LIN {X 0,Y 361.998,Z 160.89,A -85,B 0,C 180,E1 -12946.528,E2 -12946.528} C_VEL
LIN {X 0,Y 362.031,Z 160.886,A -85,B 0,C 180,E1 -12949.938,E2 -12949.938} C_VEL
LIN {X 0,Y 362.16,Z 160.873,A -85,B 0,C 180,E1 -12953.314,E2 -12953.314} C_VEL
LIN {X 0,Y 362.282,Z 160.854,A -85,B 0,C 180,E1 -12957.776,E2 -12957.776} C_VEL
LIN {X 0,Y 362.425,Z 160.836,A -85,B 0,C 180,E1 -12960,E2 -12960} C_VEL
LIN {X 0,Y 362.281,Z 160.856,A -85,B 0,C 180,E1 -12962.224,E2 -12962.224} C_VEL
LIN {X 0,Y 362.16,Z 160.875,A -85,B 0,C 180,E1 -12966.686,E2 -12966.686} C_VEL
LIN {X 0,Y 362.03,Z 160.888,A -85,B 0,C 180,E1 -12970.062,E2 -12970.062} C_VEL
LIN {X 0,Y 361.997,Z 160.891,A -85,B 0,C 180,E1 -12973.899,E2 -12973.899} C_VEL
LIN {X 0,Y 361.966,Z 160.896,A -85,B 0,C 180,E1 -12977.939,E2 -12977.939} C_VEL
LIN {X 0,Y 361.86,Z 160.908,A -85,B 0,C 180,E1 -12981.655,E2 -12981.655} C_VEL
LIN {X 0,Y 361.926,Z 160.899,A -85,B 0,C 180,E1 -12985.29,E2 -12985.29} C_VEL
LIN {X 0,Y 361.908,Z 160.905,A -85,B 0,C 180,E1 -12987.779,E2 -12987.779} C_VEL
LIN {X 0,Y 361.837,Z 160.913,A -85,B 0,C 180,E1 -12991.63,E2 -12991.63} C_VEL
LIN {X 0,Y 361.873,Z 160.907,A -85,B 0,C 180,E1 -12995.345,E2 -12995.345} C_VEL
LIN {X 0,Y 361.862,Z 160.907,A -85,B 0,C 180,E1 -12999.026,E2 -12999.026} C_VEL
LIN {X 0,Y 361.834,Z 160.911,A -85,B 0,C 180,E1 -13002.829,E2 -13002.829} C_VEL
LIN {X 0,Y 361.817,Z 160.914,A -85,B 0,C 180,E1 -13005.947,E2 -13005.947} C_VEL
LIN {X 0,Y 361.813,Z 160.918,A -85,B 0,C 180,E1 -13009.249,E2 -13009.249} C_VEL
LIN {X 0,Y 361.865,Z 160.91,A -85,B 0,C 180,E1 -13012.982,E2 -13012.982} C_VEL
LIN {X 0,Y 361.859,Z 160.909,A -85,B 0,C 180,E1 -13016.631,E2 -13016.631} C_VEL
LIN {X 0,Y 361.903,Z 160.997,A -85,B 0,C 180,E1 -13020.494,E2 -13020.494} C_VEL
LIN {X 0,Y 364.387,Z 172.887,A -85,B 0,C 180,E1 -13023.666,E2 -13023.666} C_VEL
LIN {X 0,Y 365.605,Z 180.414,A -85,B 0,C 180,E1 -13025.588,E2 -13025.588} C_VEL
LIN {X 0,Y 364.663,Z 190.236,A -85,B 0,C 180,E1 -13027.892,E2 -13027.892} C_VEL
LIN {X 0,Y 369.444,Z 217.539,A -85,B 0,C 180,E1 -13028.771,E2 -13028.771} C_VEL
LIN {X 0,Y 370.205,Z 224.641,A -85,B 0,C 180,E1 -13028.961,E2 -13028.961} C_VEL
LIN {X 0,Y 368.998,Z 298.645,A -85,B 0,C 180,E1 -13030.422,E2 -13030.422} C_VEL
LIN {X 0,Y 368.329,Z 311.846,A -85,B 0,C 180,E1 -13030.892,E2 -13030.892} C_VEL
LIN {X 0,Y 367.51,Z 323.969,A -85,B 0,C 180,E1 -13031.535,E2 -13031.535} C_VEL
LIN {X 0,Y 366.496,Z 336.205,A -85,B 0,C 180,E1 -13032.421,E2 -13032.421} C_VEL
LIN {X 0,Y 365.288,Z 347.782,A -85,B 0,C 180,E1 -13033.514,E2 -13033.514} C_VEL
LIN {X 0,Y 364.282,Z 357.893,A -85,B 0,C 180,E1 -13034.718,E2 -13034.718} C_VEL
LIN {X 0,Y 363.402,Z 366.737,A -85,B 0,C 180,E1 -13036.011,E2 -13036.011} C_VEL
LIN {X 0,Y 362.508,Z 374.603,A -85,B 0,C 180,E1 -13037.402,E2 -13037.402} C_VEL
LIN {X 0,Y 361.621,Z 382.284,A -85,B 0,C 180,E1 -13039.077,E2 -13039.077} C_VEL
LIN {X 0,Y 360.938,Z 389.371,A -85,B 0,C 180,E1 -13041.039,E2 -13041.039} C_VEL
LIN {X 0,Y 360.592,Z 394.086,A -85,B 0,C 180,E1 -13042.722,E2 -13042.722} C_VEL
LIN {X 0,Y 360.363,Z 397.689,A -85,B 0,C 180,E1 -13044.404,E2 -13044.404} C_VEL
LIN {X 0,Y 360.342,Z 399.548,A -85,B 0,C 180,E1 -13045.526,E2 -13045.526} C_VEL
LIN {X 0,Y 360.289,Z 400.941,A -85,B 0,C 180,E1 -13046.645,E2 -13046.645} C_VEL
LIN {X 0,Y 360.289,Z 402.543,A -85,B 0,C 180,E1 -13048.882,E2 -13048.882} C_VEL
LIN {X 0,Y 360.312,Z 402.757,A -85,B 0,C 180,E1 -13050,E2 -13050} C_VEL
LIN {X 0,Y 360.289,Z 402.538,A -85,B 0,C 180,E1 -13051.118,E2 -13051.118} C_VEL
LIN {X 0,Y 360.289,Z 400.931,A -85,B 0,C 180,E1 -13053.355,E2 -13053.355} C_VEL
LIN {X 0,Y 360.342,Z 399.533,A -85,B 0,C 180,E1 -13054.474,E2 -13054.474} C_VEL
LIN {X 0,Y 360.378,Z 396.969,A -85,B 0,C 180,E1 -13055.961,E2 -13055.961} C_VEL
LIN {X 0,Y 360.673,Z 392.619,A -85,B 0,C 180,E1 -13057.84,E2 -13057.84} C_VEL
LIN {X 0,Y 361.189,Z 386.507,A -85,B 0,C 180,E1 -13059.803,E2 -13059.803} C_VEL
LIN {X 0,Y 361.852,Z 379.831,A -85,B 0,C 180,E1 -13061.483,E2 -13061.483} C_VEL
LIN {X 0,Y 362.835,Z 371.552,A -85,B 0,C 180,E1 -13063.155,E2 -13063.155} C_VEL
LIN {X 0,Y 363.7,Z 363.06,A -85,B 0,C 180,E1 -13064.549,E2 -13064.549} C_VEL
LIN {X 0,Y 364.787,Z 352.569,A -85,B 0,C 180,E1 -13065.935,E2 -13065.935} C_VEL
LIN {X 0,Y 366.004,Z 340.762,A -85,B 0,C 180,E1 -13067.171,E2 -13067.171} C_VEL
LIN {X 0,Y 367.094,Z 328.878,A -85,B 0,C 180,E1 -13068.126,E2 -13068.126} C_VEL
LIN {X 0,Y 367.988,Z 316.508,A -85,B 0,C 180,E1 -13068.873,E2 -13068.873} C_VEL
LIN {X 0,Y 368.769,Z 303.791,A -85,B 0,C 180,E1 -13069.41,E2 -13069.41} C_VEL
LIN {X 0,Y 369.229,Z 290.405,A -85,B 0,C 180,E1 -13069.746,E2 -13069.746} C_VEL
LIN {X 0,Y 370.135,Z 222.324,A -85,B 0,C 180,E1 -13071.075,E2 -13071.075} C_VEL
LIN {X 0,Y 365.002,Z 192.189,A -85,B 0,C 180,E1 -13072.008,E2 -13072.008} C_VEL
LIN {X 0,Y 364.692,Z 190.305,A -85,B 0,C 180,E1 -13072.073,E2 -13072.073} C_VEL
LIN {X 0,Y 365.613,Z 180.345,A -85,B 0,C 180,E1 -13074.411,E2 -13074.411} C_VEL
LIN {X 0,Y 364.398,Z 172.814,A -85,B 0,C 180,E1 -13076.333,E2 -13076.333} C_VEL
LIN {X 0,Y 361.864,Z 160.906,A -85,B 0,C 180,E1 -13079.554,E2 -13079.554} C_VEL
LIN {X 0,Y 361.858,Z 160.909,A -85,B 0,C 180,E1 -13083.369,E2 -13083.369} C_VEL
LIN {X 0,Y 361.863,Z 160.911,A -85,B 0,C 180,E1 -13087.018,E2 -13087.018} C_VEL
LIN {X 0,Y 361.813,Z 160.919,A -85,B 0,C 180,E1 -13090.751,E2 -13090.751} C_VEL
LIN {X 0,Y 361.817,Z 160.916,A -85,B 0,C 180,E1 -13094.368,E2 -13094.368} C_VEL
LIN {X 0,Y 361.832,Z 160.91,A -85,B 0,C 180,E1 -13097.569,E2 -13097.569} C_VEL
LIN {X 0,Y 361.863,Z 160.908,A -85,B 0,C 180,E1 -13100.975,E2 -13100.975} C_VEL
LIN {X 0,Y 361.874,Z 160.908,A -85,B 0,C 180,E1 -13104.655,E2 -13104.655} C_VEL
LIN {X 0,Y 361.837,Z 160.914,A -85,B 0,C 180,E1 -13108.37,E2 -13108.37} C_VEL
LIN {X 0,Y 361.865,Z 160.906,A -85,B 0,C 180,E1 -13110.952,E2 -13110.952} C_VEL
LIN {X 0,Y 361.893,Z 160.903,A -85,B 0,C 180,E1 -13114.707,E2 -13114.707} C_VEL
LIN {X 0,Y 361.86,Z 160.909,A -85,B 0,C 180,E1 -13118.345,E2 -13118.345} C_VEL
LIN {X 0,Y 361.967,Z 160.896,A -85,B 0,C 180,E1 -13122.061,E2 -13122.061} C_VEL
LIN {X 0,Y 361.998,Z 160.891,A -85,B 0,C 180,E1 -13126.101,E2 -13126.101} C_VEL
LIN {X 0,Y 362.031,Z 160.888,A -85,B 0,C 180,E1 -13129.938,E2 -13129.938} C_VEL
LIN {X 0,Y 362.16,Z 160.874,A -85,B 0,C 180,E1 -13133.314,E2 -13133.314} C_VEL
LIN {X 0,Y 362.282,Z 160.856,A -85,B 0,C 180,E1 -13137.776,E2 -13137.776} C_VEL
LIN {X 0,Y 362.426,Z 160.836,A -85,B 0,C 180,E1 -13140,E2 -13140} C_VEL
LIN {X 0,Y 362.282,Z 160.854,A -85,B 0,C 180,E1 -13142.224,E2 -13142.224} C_VEL
LIN {X 0,Y 362.147,Z 160.874,A -85,B 0,C 180,E1 -13146.687,E2 -13146.687} C_VEL
LIN {X 0,Y 362.055,Z 160.889,A -85,B 0,C 180,E1 -13148.934,E2 -13148.934} C_VEL
LIN {X 0,Y 361.959,Z 160.896,A -85,B 0,C 180,E1 -13152.332,E2 -13152.332} C_VEL
LIN {X 0,Y 361.962,Z 160.898,A -85,B 0,C 180,E1 -13154.62,E2 -13154.62} C_VEL
LIN {X 0,Y 361.96,Z 160.895,A -85,B 0,C 180,E1 -13158.099,E2 -13158.099} C_VEL
LIN {X 0,Y 361.892,Z 160.903,A -85,B 0,C 180,E1 -13161.653,E2 -13161.653} C_VEL
LIN {X 0,Y 361.929,Z 160.898,A -85,B 0,C 180,E1 -13165.29,E2 -13165.29} C_VEL
LIN {X 0,Y 361.918,Z 160.9,A -85,B 0,C 180,E1 -13167.778,E2 -13167.778} C_VEL
LIN {X 0,Y 361.847,Z 160.908,A -85,B 0,C 180,E1 -13171.285,E2 -13171.285} C_VEL
LIN {X 0,Y 361.855,Z 160.913,A -85,B 0,C 180,E1 -13174.281,E2 -13174.281} C_VEL
LIN {X 0,Y 361.864,Z 160.906,A -85,B 0,C 180,E1 -13177.223,E2 -13177.223} C_VEL
LIN {X 0,Y 361.836,Z 160.91,A -85,B 0,C 180,E1 -13180.756,E2 -13180.756} C_VEL
LIN {X 0,Y 361.819,Z 160.914,A -85,B 0,C 180,E1 -13184.369,E2 -13184.369} C_VEL
LIN {X 0,Y 361.837,Z 160.913,A -85,B 0,C 180,E1 -13187.568,E2 -13187.568} C_VEL
LIN {X 0,Y 361.869,Z 160.906,A -85,B 0,C 180,E1 -13190.974,E2 -13190.974} C_VEL
LIN {X 0,Y 361.875,Z 160.905,A -85,B 0,C 180,E1 -13194.655,E2 -13194.655} C_VEL
LIN {X 0,Y 361.839,Z 160.91,A -85,B 0,C 180,E1 -13198.371,E2 -13198.371} C_VEL
LIN {X 0,Y 361.902,Z 160.904,A -85,B 0,C 180,E1 -13200.955,E2 -13200.955} C_VEL
LIN {X 0,Y 361.99,Z 161.002,A -85,B 0,C 180,E1 -13204.059,E2 -13204.059} C_VEL
LIN {X 0,Y 364.077,Z 171.501,A -85,B 0,C 180,E1 -13206.99,E2 -13206.99} C_VEL
LIN {X 0,Y 364.819,Z 175.438,A -85,B 0,C 180,E1 -13207.999,E2 -13207.999} C_VEL
LIN {X 0,Y 367.194,Z 184.857,A -85,B 0,C 180,E1 -13208.344,E2 -13208.344} C_VEL
LIN {X 0,Y 370.497,Z 201.339,A -85,B 0,C 180,E1 -13208.885,E2 -13208.885} C_VEL
LIN {X 0,Y 369.221,Z 281.969,A -85,B 0,C 180,E1 -13210.47,E2 -13210.47} C_VEL
LIN {X 0,Y 368.677,Z 295.427,A -85,B 0,C 180,E1 -13210.947,E2 -13210.947} C_VEL
LIN {X 0,Y 367.888,Z 308.218,A -85,B 0,C 180,E1 -13211.627,E2 -13211.627} C_VEL
LIN {X 0,Y 367.02,Z 319.572,A -85,B 0,C 180,E1 -13212.447,E2 -13212.447} C_VEL
LIN {X 0,Y 365.946,Z 331.168,A -85,B 0,C 180,E1 -13213.537,E2 -13213.537} C_VEL
LIN {X 0,Y 365.13,Z 340.627,A -85,B 0,C 180,E1 -13214.653,E2 -13214.653} C_VEL
LIN {X 0,Y 364.069,Z 350.244,A -85,B 0,C 180,E1 -13216.037,E2 -13216.037} C_VEL
LIN {X 0,Y 363.112,Z 358.121,A -85,B 0,C 180,E1 -13217.424,E2 -13217.424} C_VEL
LIN {X 0,Y 362.22,Z 365.819,A -85,B 0,C 180,E1 -13219.095,E2 -13219.095} C_VEL
LIN {X 0,Y 361.392,Z 372.884,A -85,B 0,C 180,E1 -13221.05,E2 -13221.05} C_VEL
LIN {X 0,Y 360.959,Z 377.589,A -85,B 0,C 180,E1 -13222.729,E2 -13222.729} C_VEL
LIN {X 0,Y 360.709,Z 381.189,A -85,B 0,C 180,E1 -13224.409,E2 -13224.409} C_VEL
LIN {X 0,Y 360.545,Z 383.05,A -85,B 0,C 180,E1 -13225.528,E2 -13225.528} C_VEL
LIN {X 0,Y 360.403,Z 384.452,A -85,B 0,C 180,E1 -13226.646,E2 -13226.646} C_VEL
LIN {X 0,Y 360.333,Z 386.061,A -85,B 0,C 180,E1 -13228.882,E2 -13228.882} C_VEL
LIN {X 0,Y 360.315,Z 386.294,A -85,B 0,C 180,E1 -13230,E2 -13230} C_VEL
LIN {X 0,Y 360.333,Z 386.104,A -85,B 0,C 180,E1 -13231.118,E2 -13231.118} C_VEL
LIN {X 0,Y 360.401,Z 384.552,A -85,B 0,C 180,E1 -13233.354,E2 -13233.354} C_VEL
LIN {X 0,Y 360.537,Z 383.194,A -85,B 0,C 180,E1 -13234.472,E2 -13234.472} C_VEL
LIN {X 0,Y 360.81,Z 379.409,A -85,B 0,C 180,E1 -13236.585,E2 -13236.585} C_VEL
LIN {X 0,Y 361.206,Z 374.877,A -85,B 0,C 180,E1 -13238.391,E2 -13238.391} C_VEL
LIN {X 0,Y 361.947,Z 368.434,A -85,B 0,C 180,E1 -13240.347,E2 -13240.347} C_VEL
LIN {X 0,Y 362.718,Z 361.356,A -85,B 0,C 180,E1 -13242.022,E2 -13242.022} C_VEL
LIN {X 0,Y 363.826,Z 352.532,A -85,B 0,C 180,E1 -13243.688,E2 -13243.688} C_VEL
LIN {X 0,Y 364.857,Z 343.479,A -85,B 0,C 180,E1 -13245.072,E2 -13245.072} C_VEL
LIN {X 0,Y 365.781,Z 333.461,A -85,B 0,C 180,E1 -13246.319,E2 -13246.319} C_VEL
LIN {X 0,Y 366.771,Z 322.306,A -85,B 0,C 180,E1 -13247.422,E2 -13247.422} C_VEL
LIN {X 0,Y 367.848,Z 309.786,A -85,B 0,C 180,E1 -13248.375,E2 -13248.375} C_VEL
LIN {X 0,Y 368.49,Z 299.934,A -85,B 0,C 180,E1 -13248.944,E2 -13248.944} C_VEL
LIN {X 0,Y 368.132,Z 294.363,A -85,B 0,C 180,E1 -13249.245,E2 -13249.245} C_VEL
LIN {X 0,Y 365.896,Z 285.21,A -85,B 0,C 180,E1 -13249.72,E2 -13249.72} C_VEL
LIN {X 0,Y 363.5,Z 275.916,A -85,B 0,C 180,E1 -13250.106,E2 -13250.106} C_VEL
LIN {X 0,Y 362.892,Z 270.121,A -85,B 0,C 180,E1 -13250.261,E2 -13250.261} C_VEL
LIN {X 0,Y 363.878,Z 202.414,A -85,B 0,C 180,E1 -13251.606,E2 -13251.606} C_VEL
LIN {X 0,Y 359.518,Z 180.927,A -85,B 0,C 180,E1 -13252.337,E2 -13252.337} C_VEL
LIN {X 0,Y 357.626,Z 175.212,A -85,B 0,C 180,E1 -13252.622,E2 -13252.622} C_VEL
LIN {X 0,Y 355.16,Z 162.86,A -85,B 0,C 180,E1 -13256.122,E2 -13256.122} C_VEL
LIN {X 0,Y 354.926,Z 161.775,A -85,B 0,C 180,E1 -13256.457,E2 -13256.457} C_VEL
LIN {X 0,Y 354.855,Z 161.78,A -85,B 0,C 180,E1 -13259.678,E2 -13259.678} C_VEL
LIN {X 0,Y 354.807,Z 161.786,A -85,B 0,C 180,E1 -13263.702,E2 -13263.702} C_VEL
LIN {X 0,Y 354.799,Z 161.793,A -85,B 0,C 180,E1 -13266.459,E2 -13266.459} C_VEL
LIN {X 0,Y 354.825,Z 161.783,A -85,B 0,C 180,E1 -13269.423,E2 -13269.423} C_VEL
LIN {X 0,Y 354.788,Z 161.789,A -85,B 0,C 180,E1 -13272.867,E2 -13272.867} C_VEL
LIN {X 0,Y 354.768,Z 161.796,A -85,B 0,C 180,E1 -13276.103,E2 -13276.103} C_VEL
LIN {X 0,Y 354.788,Z 161.788,A -85,B 0,C 180,E1 -13279.179,E2 -13279.179} C_VEL
LIN {X 0,Y 354.807,Z 161.787,A -85,B 0,C 180,E1 -13282.402,E2 -13282.402} C_VEL
LIN {X 0,Y 354.812,Z 161.785,A -85,B 0,C 180,E1 -13284.941,E2 -13284.941} C_VEL
LIN {X 0,Y 354.793,Z 161.788,A -85,B 0,C 180,E1 -13288.405,E2 -13288.405} C_VEL
LIN {X 0,Y 354.851,Z 161.785,A -85,B 0,C 180,E1 -13291.619,E2 -13291.619} C_VEL
LIN {X 0,Y 354.899,Z 161.775,A -85,B 0,C 180,E1 -13294.172,E2 -13294.172} C_VEL
LIN {X 0,Y 354.834,Z 161.784,A -85,B 0,C 180,E1 -13297.894,E2 -13297.894} C_VEL
LIN {X 0,Y 354.922,Z 161.772,A -85,B 0,C 180,E1 -13301.891,E2 -13301.891} C_VEL
LIN {X 0,Y 354.942,Z 161.769,A -85,B 0,C 180,E1 -13305.981,E2 -13305.981} C_VEL
LIN {X 0,Y 354.977,Z 161.765,A -85,B 0,C 180,E1 -13309.736,E2 -13309.736} C_VEL
LIN {X 0,Y 355.124,Z 161.75,A -85,B 0,C 180,E1 -13313.18,E2 -13313.18} C_VEL
LIN {X 0,Y 355.245,Z 161.73,A -85,B 0,C 180,E1 -13317.732,E2 -13317.732} C_VEL
LIN {X 0,Y 355.374,Z 161.714,A -85,B 0,C 180,E1 -13320,E2 -13320} C_VEL
LIN {X 0,Y 355.244,Z 161.733,A -85,B 0,C 180,E1 -13322.268,E2 -13322.268} C_VEL
LIN {X 0,Y 355.124,Z 161.749,A -85,B 0,C 180,E1 -13326.819,E2 -13326.819} C_VEL
LIN {X 0,Y 354.977,Z 161.768,A -85,B 0,C 180,E1 -13330.264,E2 -13330.264} C_VEL
LIN {X 0,Y 354.942,Z 161.77,A -85,B 0,C 180,E1 -13334.019,E2 -13334.019} C_VEL
LIN {X 0,Y 354.922,Z 161.776,A -85,B 0,C 180,E1 -13338.109,E2 -13338.109} C_VEL
LIN {X 0,Y 354.815,Z 161.79,A -85,B 0,C 180,E1 -13342.107,E2 -13342.107} C_VEL
LIN {X 0,Y 354.897,Z 161.777,A -85,B 0,C 180,E1 -13345.828,E2 -13345.828} C_VEL
LIN {X 0,Y 354.817,Z 161.788,A -85,B 0,C 180,E1 -13349.682,E2 -13349.682} C_VEL
LIN {X 0,Y 354.805,Z 161.791,A -85,B 0,C 180,E1 -13353.702,E2 -13353.702} C_VEL
LIN {X 0,Y 354.796,Z 161.787,A -85,B 0,C 180,E1 -13356.46,E2 -13356.46} C_VEL
LIN {X 0,Y 354.824,Z 161.787,A -85,B 0,C 180,E1 -13359.424,E2 -13359.424} C_VEL
LIN {X 0,Y 354.786,Z 161.789,A -85,B 0,C 180,E1 -13362.867,E2 -13362.867} C_VEL
LIN {X 0,Y 354.766,Z 161.791,A -85,B 0,C 180,E1 -13366.104,E2 -13366.104} C_VEL
LIN {X 0,Y 354.766,Z 161.795,A -85,B 0,C 180,E1 -13369.176,E2 -13369.176} C_VEL
LIN {X 0,Y 354.801,Z 161.787,A -85,B 0,C 180,E1 -13372.404,E2 -13372.404} C_VEL
LIN {X 0,Y 354.812,Z 161.789,A -85,B 0,C 180,E1 -13374.941,E2 -13374.941} C_VEL
LIN {X 0,Y 354.794,Z 161.789,A -85,B 0,C 180,E1 -13378.405,E2 -13378.405} C_VEL
LIN {X 0,Y 354.86,Z 161.855,A -85,B 0,C 180,E1 -13380.118,E2 -13380.118} C_VEL
LIN {X 0,Y 357.384,Z 173.967,A -85,B 0,C 180,E1 -13383.424,E2 -13383.424} C_VEL
LIN {X 0,Y 358.672,Z 181.496,A -85,B 0,C 180,E1 -13385.394,E2 -13385.394} C_VEL
LIN {X 0,Y 357.827,Z 190.115,A -85,B 0,C 180,E1 -13387.458,E2 -13387.458} C_VEL
LIN {X 0,Y 362.854,Z 218.444,A -85,B 0,C 180,E1 -13388.388,E2 -13388.388} C_VEL
LIN {X 0,Y 363.588,Z 225.102,A -85,B 0,C 180,E1 -13388.572,E2 -13388.572} C_VEL
LIN {X 0,Y 362.317,Z 298.496,A -85,B 0,C 180,E1 -13390.046,E2 -13390.046} C_VEL
LIN {X 0,Y 361.609,Z 311.692,A -85,B 0,C 180,E1 -13390.523,E2 -13390.523} C_VEL
LIN {X 0,Y 360.786,Z 323.813,A -85,B 0,C 180,E1 -13391.178,E2 -13391.178} C_VEL
LIN {X 0,Y 359.739,Z 336.048,A -85,B 0,C 180,E1 -13392.08,E2 -13392.08} C_VEL
LIN {X 0,Y 358.474,Z 347.623,A -85,B 0,C 180,E1 -13393.191,E2 -13393.191} C_VEL
LIN {X 0,Y 357.35,Z 358.451,A -85,B 0,C 180,E1 -13394.512,E2 -13394.512} C_VEL
LIN {X 0,Y 356.306,Z 368.251,A -85,B 0,C 180,E1 -13396.018,E2 -13396.018} C_VEL
LIN {X 0,Y 355.157,Z 377.175,A -85,B 0,C 180,E1 -13397.718,E2 -13397.718} C_VEL
LIN {X 0,Y 354.39,Z 384.359,A -85,B 0,C 180,E1 -13399.43,E2 -13399.43} C_VEL
LIN {X 0,Y 353.738,Z 390.902,A -85,B 0,C 180,E1 -13401.431,E2 -13401.431} C_VEL
LIN {X 0,Y 353.417,Z 395.234,A -85,B 0,C 180,E1 -13403.148,E2 -13403.148} C_VEL
LIN {X 0,Y 353.282,Z 397.527,A -85,B 0,C 180,E1 -13404.292,E2 -13404.292} C_VEL
LIN {X 0,Y 353.255,Z 399.386,A -85,B 0,C 180,E1 -13405.436,E2 -13405.436} C_VEL
LIN {X 0,Y 353.211,Z 400.78,A -85,B 0,C 180,E1 -13406.578,E2 -13406.578} C_VEL
LIN {X 0,Y 353.188,Z 402.381,A -85,B 0,C 180,E1 -13408.86,E2 -13408.86} C_VEL
LIN {X 0,Y 353.214,Z 402.595,A -85,B 0,C 180,E1 -13410,E2 -13410} C_VEL
LIN {X 0,Y 353.188,Z 402.376,A -85,B 0,C 180,E1 -13411.14,E2 -13411.14} C_VEL
LIN {X 0,Y 353.211,Z 400.769,A -85,B 0,C 180,E1 -13413.422,E2 -13413.422} C_VEL
LIN {X 0,Y 353.257,Z 399.371,A -85,B 0,C 180,E1 -13414.564,E2 -13414.564} C_VEL
LIN {X 0,Y 353.296,Z 397.076,A -85,B 0,C 180,E1 -13415.937,E2 -13415.937} C_VEL
LIN {X 0,Y 353.617,Z 392.456,A -85,B 0,C 180,E1 -13417.997,E2 -13417.997} C_VEL
LIN {X 0,Y 354.17,Z 386.343,A -85,B 0,C 180,E1 -13419.999,E2 -13419.999} C_VEL
LIN {X 0,Y 354.875,Z 379.667,A -85,B 0,C 180,E1 -13421.712,E2 -13421.712} C_VEL
LIN {X 0,Y 355.903,Z 371.387,A -85,B 0,C 180,E1 -13423.416,E2 -13423.416} C_VEL
LIN {X 0,Y 356.81,Z 362.895,A -85,B 0,C 180,E1 -13424.836,E2 -13424.836} C_VEL
LIN {X 0,Y 357.934,Z 352.403,A -85,B 0,C 180,E1 -13426.248,E2 -13426.248} C_VEL
LIN {X 0,Y 359.193,Z 340.595,A -85,B 0,C 180,E1 -13427.507,E2 -13427.507} C_VEL
LIN {X 0,Y 360.344,Z 328.71,A -85,B 0,C 180,E1 -13428.478,E2 -13428.478} C_VEL
LIN {X 0,Y 361.294,Z 316.339,A -85,B 0,C 180,E1 -13429.237,E2 -13429.237} C_VEL
LIN {X 0,Y 362.103,Z 303.619,A -85,B 0,C 180,E1 -13429.782,E2 -13429.782} C_VEL
LIN {X 0,Y 362.564,Z 290.223,A -85,B 0,C 180,E1 -13430.125,E2 -13430.125} C_VEL
LIN {X 0,Y 363.525,Z 223.338,A -85,B 0,C 180,E1 -13431.453,E2 -13431.453} C_VEL
LIN {X 0,Y 358.215,Z 192.075,A -85,B 0,C 180,E1 -13432.446,E2 -13432.446} C_VEL
LIN {X 0,Y 357.856,Z 190.155,A -85,B 0,C 180,E1 -13432.514,E2 -13432.514} C_VEL
LIN {X 0,Y 358.679,Z 181.422,A -85,B 0,C 180,E1 -13434.606,E2 -13434.606} C_VEL
LIN {X 0,Y 356.842,Z 171.032,A -85,B 0,C 180,E1 -13437.339,E2 -13437.339} C_VEL
LIN {X 0,Y 354.813,Z 161.782,A -85,B 0,C 180,E1 -13439.927,E2 -13439.927} C_VEL
LIN {X 0,Y 354.807,Z 161.786,A -85,B 0,C 180,E1 -13443.702,E2 -13443.702} C_VEL
LIN {X 0,Y 354.794,Z 161.79,A -85,B 0,C 180,E1 -13446.46,E2 -13446.46} C_VEL
LIN {X 0,Y 354.768,Z 161.791,A -85,B 0,C 180,E1 -13449.412,E2 -13449.412} C_VEL
LIN {X 0,Y 354.785,Z 161.792,A -85,B 0,C 180,E1 -13452.866,E2 -13452.866} C_VEL
LIN {X 0,Y 354.767,Z 161.793,A -85,B 0,C 180,E1 -13456.103,E2 -13456.103} C_VEL
LIN {X 0,Y 354.782,Z 161.789,A -85,B 0,C 180,E1 -13459.178,E2 -13459.178} C_VEL
LIN {X 0,Y 354.805,Z 161.791,A -85,B 0,C 180,E1 -13462.403,E2 -13462.403} C_VEL
LIN {X 0,Y 354.811,Z 161.786,A -85,B 0,C 180,E1 -13464.941,E2 -13464.941} C_VEL
LIN {X 0,Y 354.793,Z 161.791,A -85,B 0,C 180,E1 -13468.405,E2 -13468.405} C_VEL
LIN {X 0,Y 354.802,Z 161.788,A -85,B 0,C 180,E1 -13471.615,E2 -13471.615} C_VEL
LIN {X 0,Y 354.851,Z 161.781,A -85,B 0,C 180,E1 -13475.423,E2 -13475.423} C_VEL
LIN {X 0,Y 354.826,Z 161.783,A -85,B 0,C 180,E1 -13479.113,E2 -13479.113} C_VEL
LIN {X 0,Y 354.898,Z 161.774,A -85,B 0,C 180,E1 -13482.72,E2 -13482.72} C_VEL
LIN {X 0,Y 354.951,Z 161.768,A -85,B 0,C 180,E1 -13486.255,E2 -13486.255} C_VEL
LIN {X 0,Y 354.977,Z 161.768,A -85,B 0,C 180,E1 -13489.736,E2 -13489.736} C_VEL
LIN {X 0,Y 355.124,Z 161.749,A -85,B 0,C 180,E1 -13493.181,E2 -13493.181} C_VEL
LIN {X 0,Y 355.245,Z 161.733,A -85,B 0,C 180,E1 -13497.732,E2 -13497.732} C_VEL
LIN {X 0,Y 355.375,Z 161.715,A -85,B 0,C 180,E1 -13500,E2 -13500} C_VEL
LIN {X 0,Y 355.245,Z 161.731,A -85,B 0,C 180,E1 -13502.268,E2 -13502.268} C_VEL
LIN {X 0,Y 355.113,Z 161.751,A -85,B 0,C 180,E1 -13506.82,E2 -13506.82} C_VEL
LIN {X 0,Y 355.004,Z 161.765,A -85,B 0,C 180,E1 -13509.113,E2 -13509.113} C_VEL
LIN {X 0,Y 354.921,Z 161.774,A -85,B 0,C 180,E1 -13512.581,E2 -13512.581} C_VEL
LIN {X 0,Y 354.89,Z 161.776,A -85,B 0,C 180,E1 -13516.096,E2 -13516.096} C_VEL
LIN {X 0,Y 354.906,Z 161.776,A -85,B 0,C 180,E1 -13518.472,E2 -13518.472} C_VEL
LIN {X 0,Y 354.835,Z 161.784,A -85,B 0,C 180,E1 -13522.106,E2 -13522.106} C_VEL
LIN {X 0,Y 354.9,Z 161.775,A -85,B 0,C 180,E1 -13525.828,E2 -13525.828} C_VEL
LIN {X 0,Y 354.854,Z 161.78,A -85,B 0,C 180,E1 -13529.679,E2 -13529.679} C_VEL
LIN {X 0,Y 354.806,Z 161.787,A -85,B 0,C 180,E1 -13533.702,E2 -13533.702} C_VEL
LIN {X 0,Y 354.799,Z 161.789,A -85,B 0,C 180,E1 -13536.46,E2 -13536.46} C_VEL
LIN {X 0,Y 354.825,Z 161.784,A -85,B 0,C 180,E1 -13539.424,E2 -13539.424} C_VEL
LIN {X 0,Y 354.789,Z 161.788,A -85,B 0,C 180,E1 -13542.867,E2 -13542.867} C_VEL
LIN {X 0,Y 354.769,Z 161.794,A -85,B 0,C 180,E1 -13546.104,E2 -13546.104} C_VEL
LIN {X 0,Y 354.789,Z 161.789,A -85,B 0,C 180,E1 -13549.179,E2 -13549.179} C_VEL
LIN {X 0,Y 354.808,Z 161.786,A -85,B 0,C 180,E1 -13552.403,E2 -13552.403} C_VEL
LIN {X 0,Y 354.813,Z 161.786,A -85,B 0,C 180,E1 -13554.941,E2 -13554.941} C_VEL
LIN {X 0,Y 354.795,Z 161.788,A -85,B 0,C 180,E1 -13558.405,E2 -13558.405} C_VEL
LIN {X 0,Y 354.853,Z 161.785,A -85,B 0,C 180,E1 -13561.619,E2 -13561.619} C_VEL
LIN {X 0,Y 354.934,Z 161.879,A -85,B 0,C 180,E1 -13563.702,E2 -13563.702} C_VEL
LIN {X 0,Y 357.125,Z 172.824,A -85,B 0,C 180,E1 -13566.822,E2 -13566.822} C_VEL
LIN {X 0,Y 357.628,Z 175.429,A -85,B 0,C 180,E1 -13567.528,E2 -13567.528} C_VEL
LIN {X 0,Y 359.812,Z 182.347,A -85,B 0,C 180,E1 -13567.819,E2 -13567.819} C_VEL
LIN {X 0,Y 363.937,Z 203.054,A -85,B 0,C 180,E1 -13568.518,E2 -13568.518} C_VEL
LIN {X 0,Y 362.557,Z 282.149,A -85,B 0,C 180,E1 -13570.096,E2 -13570.096} C_VEL
LIN {X 0,Y 361.989,Z 295.599,A -85,B 0,C 180,E1 -13570.581,E2 -13570.581} C_VEL
LIN {X 0,Y 361.173,Z 308.388,A -85,B 0,C 180,E1 -13571.272,E2 -13571.272} C_VEL
LIN {X 0,Y 360.269,Z 319.739,A -85,B 0,C 180,E1 -13572.107,E2 -13572.107} C_VEL
LIN {X 0,Y 359.271,Z 330.239,A -85,B 0,C 180,E1 -13573.098,E2 -13573.098} C_VEL
LIN {X 0,Y 358.342,Z 339.728,A -85,B 0,C 180,E1 -13574.209,E2 -13574.209} C_VEL
LIN {X 0,Y 357.386,Z 348.634,A -85,B 0,C 180,E1 -13575.479,E2 -13575.479} C_VEL
LIN {X 0,Y 356.162,Z 358.286,A -85,B 0,C 180,E1 -13577.174,E2 -13577.174} C_VEL
LIN {X 0,Y 355.244,Z 365.984,A -85,B 0,C 180,E1 -13578.879,E2 -13578.879} C_VEL
LIN {X 0,Y 354.389,Z 373.048,A -85,B 0,C 180,E1 -13580.871,E2 -13580.871} C_VEL
LIN {X 0,Y 353.92,Z 377.752,A -85,B 0,C 180,E1 -13582.584,E2 -13582.584} C_VEL
LIN {X 0,Y 353.642,Z 381.352,A -85,B 0,C 180,E1 -13584.297,E2 -13584.297} C_VEL
LIN {X 0,Y 353.484,Z 383.213,A -85,B 0,C 180,E1 -13585.439,E2 -13585.439} C_VEL
LIN {X 0,Y 353.325,Z 384.614,A -85,B 0,C 180,E1 -13586.579,E2 -13586.579} C_VEL
LIN {X 0,Y 353.235,Z 386.223,A -85,B 0,C 180,E1 -13588.86,E2 -13588.86} C_VEL
LIN {X 0,Y 353.217,Z 386.456,A -85,B 0,C 180,E1 -13590,E2 -13590} C_VEL
LIN {X 0,Y 353.235,Z 386.266,A -85,B 0,C 180,E1 -13591.14,E2 -13591.14} C_VEL
LIN {X 0,Y 353.322,Z 384.714,A -85,B 0,C 180,E1 -13593.421,E2 -13593.421} C_VEL
LIN {X 0,Y 353.475,Z 383.355,A -85,B 0,C 180,E1 -13594.562,E2 -13594.562} C_VEL
LIN {X 0,Y 353.739,Z 379.844,A -85,B 0,C 180,E1 -13596.59,E2 -13596.59} C_VEL
LIN {X 0,Y 354.187,Z 375.038,A -85,B 0,C 180,E1 -13598.558,E2 -13598.558} C_VEL
LIN {X 0,Y 354.934,Z 368.595,A -85,B 0,C 180,E1 -13600.554,E2 -13600.554} C_VEL
LIN {X 0,Y 355.759,Z 361.516,A -85,B 0,C 180,E1 -13602.261,E2 -13602.261} C_VEL
LIN {X 0,Y 356.945,Z 352.691,A -85,B 0,C 180,E1 -13603.957,E2 -13603.957} C_VEL
LIN {X 0,Y 358.002,Z 343.638,A -85,B 0,C 180,E1 -13605.368,E2 -13605.368} C_VEL
LIN {X 0,Y 358.928,Z 333.995,A -85,B 0,C 180,E1 -13606.596,E2 -13606.596} C_VEL
LIN {X 0,Y 360.005,Z 322.463,A -85,B 0,C 180,E1 -13607.76,E2 -13607.76} C_VEL
LIN {X 0,Y 361.137,Z 309.941,A -85,B 0,C 180,E1 -13608.729,E2 -13608.729} C_VEL
LIN {X 0,Y 361.915,Z 297.04,A -85,B 0,C 180,E1 -13609.46,E2 -13609.46} C_VEL
LIN {X 0,Y 362.514,Z 284.323,A -85,B 0,C 180,E1 -13609.943,E2 -13609.943} C_VEL
LIN {X 0,Y 362.892,Z 270.121,A -85,B 0,C 180,E1 -13610.261,E2 -13610.261} C_VEL
LIN {X 0,Y 362.265,Z 264.318,A -85,B 0,C 180,E1 -13610.418,E2 -13610.418} C_VEL
LIN {X 0,Y 357.184,Z 245.65,A -85,B 0,C 180,E1 -13611.118,E2 -13611.118} C_VEL
LIN {X 0,Y 356.761,Z 239.844,A -85,B 0,C 180,E1 -13611.267,E2 -13611.267} C_VEL
LIN {X 0,Y 357.316,Z 203.475,A -85,B 0,C 180,E1 -13612.003,E2 -13612.003} C_VEL
LIN {X 0,Y 353.164,Z 182.998,A -85,B 0,C 180,E1 -13612.72,E2 -13612.72} C_VEL
LIN {X 0,Y 350.446,Z 175.432,A -85,B 0,C 180,E1 -13613.097,E2 -13613.097} C_VEL
LIN {X 0,Y 348.181,Z 164.168,A -85,B 0,C 180,E1 -13616.364,E2 -13616.364} C_VEL
LIN {X 0,Y 347.853,Z 162.657,A -85,B 0,C 180,E1 -13616.856,E2 -13616.856} C_VEL
LIN {X 0,Y 347.765,Z 162.667,A -85,B 0,C 180,E1 -13620.346,E2 -13620.346} C_VEL
LIN {X 0,Y 347.745,Z 162.669,A -85,B 0,C 180,E1 -13624.464,E2 -13624.464} C_VEL
LIN {X 0,Y 347.774,Z 162.664,A -85,B 0,C 180,E1 -13627.988,E2 -13627.988} C_VEL
LIN {X 0,Y 347.751,Z 162.666,A -85,B 0,C 180,E1 -13631.83,E2 -13631.83} C_VEL
LIN {X 0,Y 347.707,Z 162.67,A -85,B 0,C 180,E1 -13635.026,E2 -13635.026} C_VEL
LIN {X 0,Y 347.75,Z 162.667,A -85,B 0,C 180,E1 -13638.397,E2 -13638.397} C_VEL
LIN {X 0,Y 347.773,Z 162.666,A -85,B 0,C 180,E1 -13642.011,E2 -13642.011} C_VEL
LIN {X 0,Y 347.744,Z 162.668,A -85,B 0,C 180,E1 -13645.536,E2 -13645.536} C_VEL
LIN {X 0,Y 347.763,Z 162.668,A -85,B 0,C 180,E1 -13649.653,E2 -13649.653} C_VEL
LIN {X 0,Y 347.851,Z 162.651,A -85,B 0,C 180,E1 -13652.744,E2 -13652.744} C_VEL
LIN {X 0,Y 347.788,Z 162.66,A -85,B 0,C 180,E1 -13656.162,E2 -13656.162} C_VEL
LIN {X 0,Y 347.817,Z 162.658,A -85,B 0,C 180,E1 -13659.909,E2 -13659.909} C_VEL
LIN {X 0,Y 347.866,Z 162.65,A -85,B 0,C 180,E1 -13662.359,E2 -13662.359} C_VEL
LIN {X 0,Y 347.897,Z 162.646,A -85,B 0,C 180,E1 -13665.971,E2 -13665.971} C_VEL
LIN {X 0,Y 347.928,Z 162.644,A -85,B 0,C 180,E1 -13669.525,E2 -13669.525} C_VEL
LIN {X 0,Y 348.091,Z 162.627,A -85,B 0,C 180,E1 -13673.042,E2 -13673.042} C_VEL
LIN {X 0,Y 348.207,Z 162.607,A -85,B 0,C 180,E1 -13677.686,E2 -13677.686} C_VEL
LIN {X 0,Y 348.324,Z 162.592,A -85,B 0,C 180,E1 -13680,E2 -13680} C_VEL
LIN {X 0,Y 348.207,Z 162.61,A -85,B 0,C 180,E1 -13682.313,E2 -13682.313} C_VEL
LIN {X 0,Y 348.091,Z 162.624,A -85,B 0,C 180,E1 -13686.958,E2 -13686.958} C_VEL
LIN {X 0,Y 347.927,Z 162.648,A -85,B 0,C 180,E1 -13690.474,E2 -13690.474} C_VEL
LIN {X 0,Y 347.898,Z 162.648,A -85,B 0,C 180,E1 -13694.15,E2 -13694.15} C_VEL
LIN {X 0,Y 347.89,Z 162.651,A -85,B 0,C 180,E1 -13698.29,E2 -13698.29} C_VEL
LIN {X 0,Y 347.766,Z 162.664,A -85,B 0,C 180,E1 -13701.626,E2 -13701.626} C_VEL
LIN {X 0,Y 347.81,Z 162.656,A -85,B 0,C 180,E1 -13705.109,E2 -13705.109} C_VEL
LIN {X 0,Y 347.807,Z 162.661,A -85,B 0,C 180,E1 -13707.694,E2 -13707.694} C_VEL
LIN {X 0,Y 347.748,Z 162.666,A -85,B 0,C 180,E1 -13710.348,E2 -13710.348} C_VEL
LIN {X 0,Y 347.747,Z 162.668,A -85,B 0,C 180,E1 -13714.044,E2 -13714.044} C_VEL
LIN {X 0,Y 347.76,Z 162.666,A -85,B 0,C 180,E1 -13717.321,E2 -13717.321} C_VEL
LIN {X 0,Y 347.728,Z 162.668,A -85,B 0,C 180,E1 -13720.298,E2 -13720.298} C_VEL
LIN {X 0,Y 347.722,Z 162.673,A -85,B 0,C 180,E1 -13723.408,E2 -13723.408} C_VEL
LIN {X 0,Y 347.724,Z 162.668,A -85,B 0,C 180,E1 -13726.687,E2 -13726.687} C_VEL
LIN {X 0,Y 347.701,Z 162.671,A -85,B 0,C 180,E1 -13730.183,E2 -13730.183} C_VEL
LIN {X 0,Y 347.757,Z 162.665,A -85,B 0,C 180,E1 -13732.679,E2 -13732.679} C_VEL
LIN {X 0,Y 347.749,Z 162.666,A -85,B 0,C 180,E1 -13735.956,E2 -13735.956} C_VEL
LIN {X 0,Y 347.803,Z 162.711,A -85,B 0,C 180,E1 -13739.724,E2 -13739.724} C_VEL
LIN {X 0,Y 350.384,Z 175.046,A -85,B 0,C 180,E1 -13743.173,E2 -13743.173} C_VEL
LIN {X 0,Y 351.733,Z 182.576,A -85,B 0,C 180,E1 -13745.191,E2 -13745.191} C_VEL
LIN {X 0,Y 351.031,Z 189.984,A -85,B 0,C 180,E1 -13747.005,E2 -13747.005} C_VEL
LIN {X 0,Y 356.277,Z 219.455,A -85,B 0,C 180,E1 -13747.993,E2 -13747.993} C_VEL
LIN {X 0,Y 356.974,Z 226.191,A -85,B 0,C 180,E1 -13748.181,E2 -13748.181} C_VEL
LIN {X 0,Y 355.656,Z 298.347,A -85,B 0,C 180,E1 -13749.656,E2 -13749.656} C_VEL
LIN {X 0,Y 354.93,Z 311.538,A -85,B 0,C 180,E1 -13750.141,E2 -13750.141} C_VEL
LIN {X 0,Y 353.987,Z 324.773,A -85,B 0,C 180,E1 -13750.878,E2 -13750.878} C_VEL
LIN {X 0,Y 352.986,Z 335.89,A -85,B 0,C 180,E1 -13751.725,E2 -13751.725} C_VEL
LIN {X 0,Y 351.671,Z 347.464,A -85,B 0,C 180,E1 -13752.856,E2 -13752.856} C_VEL
LIN {X 0,Y 350.469,Z 358.4,A -85,B 0,C 180,E1 -13754.215,E2 -13754.215} C_VEL
LIN {X 0,Y 349.385,Z 368.09,A -85,B 0,C 180,E1 -13755.735,E2 -13755.735} C_VEL
LIN {X 0,Y 348.208,Z 377.014,A -85,B 0,C 180,E1 -13757.469,E2 -13757.469} C_VEL
LIN {X 0,Y 347.401,Z 384.198,A -85,B 0,C 180,E1 -13759.215,E2 -13759.215} C_VEL
LIN {X 0,Y 346.693,Z 390.741,A -85,B 0,C 180,E1 -13761.255,E2 -13761.255} C_VEL
LIN {X 0,Y 346.343,Z 395.072,A -85,B 0,C 180,E1 -13763.007,E2 -13763.007} C_VEL
LIN {X 0,Y 346.201,Z 397.365,A -85,B 0,C 180,E1 -13764.174,E2 -13764.174} C_VEL
LIN {X 0,Y 346.154,Z 399.224,A -85,B 0,C 180,E1 -13765.342,E2 -13765.342} C_VEL
LIN {X 0,Y 346.134,Z 400.618,A -85,B 0,C 180,E1 -13766.508,E2 -13766.508} C_VEL
LIN {X 0,Y 346.089,Z 402.219,A -85,B 0,C 180,E1 -13768.836,E2 -13768.836} C_VEL
LIN {X 0,Y 346.116,Z 402.433,A -85,B 0,C 180,E1 -13770,E2 -13770} C_VEL
LIN {X 0,Y 346.089,Z 402.213,A -85,B 0,C 180,E1 -13771.164,E2 -13771.164} C_VEL
LIN {X 0,Y 346.134,Z 400.607,A -85,B 0,C 180,E1 -13773.492,E2 -13773.492} C_VEL
LIN {X 0,Y 346.155,Z 399.207,A -85,B 0,C 180,E1 -13774.658,E2 -13774.658} C_VEL
LIN {X 0,Y 346.26,Z 396.269,A -85,B 0,C 180,E1 -13776.409,E2 -13776.409} C_VEL
LIN {X 0,Y 346.557,Z 392.292,A -85,B 0,C 180,E1 -13778.161,E2 -13778.161} C_VEL
LIN {X 0,Y 347.142,Z 386.179,A -85,B 0,C 180,E1 -13780.204,E2 -13780.204} C_VEL
LIN {X 0,Y 347.895,Z 379.502,A -85,B 0,C 180,E1 -13781.95,E2 -13781.95} C_VEL
LIN {X 0,Y 348.979,Z 371.222,A -85,B 0,C 180,E1 -13783.688,E2 -13783.688} C_VEL
LIN {X 0,Y 350.048,Z 361.571,A -85,B 0,C 180,E1 -13785.307,E2 -13785.307} C_VEL
LIN {X 0,Y 351.22,Z 351.06,A -85,B 0,C 180,E1 -13786.717,E2 -13786.717} C_VEL
LIN {X 0,Y 352.413,Z 340.428,A -85,B 0,C 180,E1 -13787.855,E2 -13787.855} C_VEL
LIN {X 0,Y 353.605,Z 328.541,A -85,B 0,C 180,E1 -13788.843,E2 -13788.843} C_VEL
LIN {X 0,Y 354.505,Z 317.471,A -85,B 0,C 180,E1 -13789.545,E2 -13789.545} C_VEL
LIN {X 0,Y 355.361,Z 304.366,A -85,B 0,C 180,E1 -13790.136,E2 -13790.136} C_VEL
LIN {X 0,Y 355.877,Z 291.83,A -85,B 0,C 180,E1 -13790.482,E2 -13790.482} C_VEL
LIN {X 0,Y 356.85,Z 223.891,A -85,B 0,C 180,E1 -13791.859,E2 -13791.859} C_VEL
LIN {X 0,Y 352.038,Z 195.356,A -85,B 0,C 180,E1 -13792.787,E2 -13792.787} C_VEL
LIN {X 0,Y 351.034,Z 189.871,A -85,B 0,C 180,E1 -13793.005,E2 -13793.005} C_VEL
LIN {X 0,Y 351.73,Z 182.499,A -85,B 0,C 180,E1 -13794.81,E2 -13794.81} C_VEL
LIN {X 0,Y 349.905,Z 172.452,A -85,B 0,C 180,E1 -13797.514,E2 -13797.514} C_VEL
LIN {X 0,Y 347.798,Z 162.657,A -85,B 0,C 180,E1 -13800.297,E2 -13800.297} C_VEL
LIN {X 0,Y 347.743,Z 162.668,A -85,B 0,C 180,E1 -13804.464,E2 -13804.464} C_VEL
LIN {X 0,Y 347.763,Z 162.664,A -85,B 0,C 180,E1 -13807.986,E2 -13807.986} C_VEL
LIN {X 0,Y 347.744,Z 162.666,A -85,B 0,C 180,E1 -13811.831,E2 -13811.831} C_VEL
LIN {X 0,Y 347.705,Z 162.672,A -85,B 0,C 180,E1 -13815.027,E2 -13815.027} C_VEL
LIN {X 0,Y 347.747,Z 162.67,A -85,B 0,C 180,E1 -13818.398,E2 -13818.398} C_VEL
LIN {X 0,Y 347.771,Z 162.665,A -85,B 0,C 180,E1 -13822.012,E2 -13822.012} C_VEL
LIN {X 0,Y 347.744,Z 162.666,A -85,B 0,C 180,E1 -13825.536,E2 -13825.536} C_VEL
LIN {X 0,Y 347.745,Z 162.67,A -85,B 0,C 180,E1 -13828.3,E2 -13828.3} C_VEL
LIN {X 0,Y 347.746,Z 162.665,A -85,B 0,C 180,E1 -13830.985,E2 -13830.985} C_VEL
LIN {X 0,Y 347.785,Z 162.66,A -85,B 0,C 180,E1 -13834.889,E2 -13834.889} C_VEL
LIN {X 0,Y 347.78,Z 162.661,A -85,B 0,C 180,E1 -13838.669,E2 -13838.669} C_VEL
LIN {X 0,Y 347.866,Z 162.65,A -85,B 0,C 180,E1 -13842.359,E2 -13842.359} C_VEL
LIN {X 0,Y 347.897,Z 162.649,A -85,B 0,C 180,E1 -13845.971,E2 -13845.971} C_VEL
LIN {X 0,Y 347.928,Z 162.648,A -85,B 0,C 180,E1 -13849.526,E2 -13849.526} C_VEL
LIN {X 0,Y 348.09,Z 162.624,A -85,B 0,C 180,E1 -13853.042,E2 -13853.042} C_VEL
LIN {X 0,Y 348.207,Z 162.609,A -85,B 0,C 180,E1 -13857.687,E2 -13857.687} C_VEL
LIN {X 0,Y 348.325,Z 162.592,A -85,B 0,C 180,E1 -13860,E2 -13860} C_VEL
LIN {X 0,Y 348.208,Z 162.608,A -85,B 0,C 180,E1 -13862.314,E2 -13862.314} C_VEL
LIN {X 0,Y 348.081,Z 162.628,A -85,B 0,C 180,E1 -13866.958,E2 -13866.958} C_VEL
LIN {X 0,Y 347.944,Z 162.643,A -85,B 0,C 180,E1 -13869.299,E2 -13869.299} C_VEL
LIN {X 0,Y 347.89,Z 162.652,A -85,B 0,C 180,E1 -13872.84,E2 -13872.84} C_VEL
LIN {X 0,Y 347.839,Z 162.656,A -85,B 0,C 180,E1 -13876.431,E2 -13876.431} C_VEL
LIN {X 0,Y 347.856,Z 162.655,A -85,B 0,C 180,E1 -13878.86,E2 -13878.86} C_VEL
LIN {X 0,Y 347.774,Z 162.666,A -85,B 0,C 180,E1 -13882.579,E2 -13882.579} C_VEL
LIN {X 0,Y 347.812,Z 162.658,A -85,B 0,C 180,E1 -13885.109,E2 -13885.109} C_VEL
LIN {X 0,Y 347.811,Z 162.657,A -85,B 0,C 180,E1 -13887.694,E2 -13887.694} C_VEL
LIN {X 0,Y 347.764,Z 162.668,A -85,B 0,C 180,E1 -13890.347,E2 -13890.347} C_VEL
LIN {X 0,Y 347.745,Z 162.668,A -85,B 0,C 180,E1 -13894.464,E2 -13894.464} C_VEL
LIN {X 0,Y 347.774,Z 162.667,A -85,B 0,C 180,E1 -13897.989,E2 -13897.989} C_VEL
LIN {X 0,Y 347.751,Z 162.669,A -85,B 0,C 180,E1 -13901.83,E2 -13901.83} C_VEL
LIN {X 0,Y 347.707,Z 162.67,A -85,B 0,C 180,E1 -13905.027,E2 -13905.027} C_VEL
LIN {X 0,Y 347.751,Z 162.665,A -85,B 0,C 180,E1 -13908.397,E2 -13908.397} C_VEL
LIN {X 0,Y 347.774,Z 162.665,A -85,B 0,C 180,E1 -13912.012,E2 -13912.012} C_VEL
LIN {X 0,Y 347.746,Z 162.672,A -85,B 0,C 180,E1 -13915.536,E2 -13915.536} C_VEL
LIN {X 0,Y 347.766,Z 162.668,A -85,B 0,C 180,E1 -13919.654,E2 -13919.654} C_VEL
LIN {X 0,Y 347.898,Z 162.821,A -85,B 0,C 180,E1 -13923.348,E2 -13923.348} C_VEL
LIN {X 0,Y 349.983,Z 172.995,A -85,B 0,C 180,E1 -13926.321,E2 -13926.321} C_VEL
LIN {X 0,Y 350.497,Z 175.787,A -85,B 0,C 180,E1 -13927.048,E2 -13927.048} C_VEL
LIN {X 0,Y 353.35,Z 183.843,A -85,B 0,C 180,E1 -13927.42,E2 -13927.42} C_VEL
LIN {X 0,Y 357.36,Z 204.145,A -85,B 0,C 180,E1 -13928.121,E2 -13928.121} C_VEL
LIN {X 0,Y 355.892,Z 282.329,A -85,B 0,C 180,E1 -13929.707,E2 -13929.707} C_VEL
LIN {X 0,Y 355.316,Z 295.772,A -85,B 0,C 180,E1 -13930.201,E2 -13930.201} C_VEL
LIN {X 0,Y 354.476,Z 308.558,A -85,B 0,C 180,E1 -13930.905,E2 -13930.905} C_VEL
LIN {X 0,Y 353.52,Z 319.907,A -85,B 0,C 180,E1 -13931.753,E2 -13931.753} C_VEL
LIN {X 0,Y 352.321,Z 331.823,A -85,B 0,C 180,E1 -13932.919,E2 -13932.919} C_VEL
LIN {X 0,Y 351.307,Z 342.183,A -85,B 0,C 180,E1 -13934.205,E2 -13934.205} C_VEL
LIN {X 0,Y 350.316,Z 350.574,A -85,B 0,C 180,E1 -13935.477,E2 -13935.477} C_VEL
LIN {X 0,Y 349.234,Z 358.451,A -85,B 0,C 180,E1 -13936.915,E2 -13936.915} C_VEL
LIN {X 0,Y 348.257,Z 366.148,A -85,B 0,C 180,E1 -13938.652,E2 -13938.652} C_VEL
LIN {X 0,Y 347.37,Z 373.212,A -85,B 0,C 180,E1 -13940.685,E2 -13940.685} C_VEL
LIN {X 0,Y 346.861,Z 377.916,A -85,B 0,C 180,E1 -13942.432,E2 -13942.432} C_VEL
LIN {X 0,Y 346.562,Z 381.515,A -85,B 0,C 180,E1 -13944.18,E2 -13944.18} C_VEL
LIN {X 0,Y 346.425,Z 383.375,A -85,B 0,C 180,E1 -13945.345,E2 -13945.345} C_VEL
LIN {X 0,Y 346.251,Z 384.777,A -85,B 0,C 180,E1 -13946.509,E2 -13946.509} C_VEL
LIN {X 0,Y 346.137,Z 386.386,A -85,B 0,C 180,E1 -13948.837,E2 -13948.837} C_VEL
LIN {X 0,Y 346.12,Z 386.618,A -85,B 0,C 180,E1 -13950,E2 -13950} C_VEL
LIN {X 0,Y 346.137,Z 386.428,A -85,B 0,C 180,E1 -13951.163,E2 -13951.163} C_VEL
LIN {X 0,Y 346.248,Z 384.875,A -85,B 0,C 180,E1 -13953.491,E2 -13953.491} C_VEL
LIN {X 0,Y 346.416,Z 383.516,A -85,B 0,C 180,E1 -13954.655,E2 -13954.655} C_VEL
LIN {X 0,Y 346.664,Z 380.289,A -85,B 0,C 180,E1 -13956.589,E2 -13956.589} C_VEL
LIN {X 0,Y 347.158,Z 375.199,A -85,B 0,C 180,E1 -13958.733,E2 -13958.733} C_VEL
LIN {X 0,Y 347.939,Z 368.756,A -85,B 0,C 180,E1 -13960.768,E2 -13960.768} C_VEL
LIN {X 0,Y 348.812,Z 361.676,A -85,B 0,C 180,E1 -13962.509,E2 -13962.509} C_VEL
LIN {X 0,Y 350.055,Z 352.851,A -85,B 0,C 180,E1 -13964.237,E2 -13964.237} C_VEL
LIN {X 0,Y 351.123,Z 344.122,A -85,B 0,C 180,E1 -13965.627,E2 -13965.627} C_VEL
LIN {X 0,Y 352.168,Z 333.777,A -85,B 0,C 180,E1 -13966.969,E2 -13966.969} C_VEL
LIN {X 0,Y 353.266,Z 322.619,A -85,B 0,C 180,E1 -13968.11,E2 -13968.11} C_VEL
LIN {X 0,Y 354.444,Z 310.096,A -85,B 0,C 180,E1 -13969.097,E2 -13969.097} C_VEL
LIN {X 0,Y 355.247,Z 297.191,A -85,B 0,C 180,E1 -13969.841,E2 -13969.841} C_VEL
LIN {X 0,Y 355.862,Z 284.469,A -85,B 0,C 180,E1 -13970.332,E2 -13970.332} C_VEL
LIN {X 0,Y 356.479,Z 255.198,A -85,B 0,C 180,E1 -13970.96,E2 -13970.96} C_VEL
LIN {X 0,Y 356.761,Z 239.844,A -85,B 0,C 180,E1 -13971.267,E2 -13971.267} C_VEL
LIN {X 0,Y 356.36,Z 234.04,A -85,B 0,C 180,E1 -13971.416,E2 -13971.416} C_VEL
LIN {X 0,Y 351.824,Z 217.256,A -85,B 0,C 180,E1 -13972.07,E2 -13972.07} C_VEL
LIN {X 0,Y 350.826,Z 211.523,A -85,B 0,C 180,E1 -13972.261,E2 -13972.261} C_VEL
LIN {X 0,Y 350.71,Z 209.572,A -85,B 0,C 180,E1 -13972.311,E2 -13972.311} C_VEL
LIN {X 0,Y 350.609,Z 203.576,A -85,B 0,C 180,E1 -13972.448,E2 -13972.448} C_VEL
LIN {X 0,Y 346.752,Z 185.026,A -85,B 0,C 180,E1 -13973.122,E2 -13973.122} C_VEL
LIN {X 0,Y 343.27,Z 175.671,A -85,B 0,C 180,E1 -13973.591,E2 -13973.591} C_VEL
LIN {X 0,Y 341.246,Z 165.48,A -85,B 0,C 180,E1 -13976.612,E2 -13976.612} C_VEL
LIN {X 0,Y 340.815,Z 163.532,A -85,B 0,C 180,E1 -13977.25,E2 -13977.25} C_VEL
LIN {X 0,Y 340.765,Z 163.537,A -85,B 0,C 180,E1 -13979.978,E2 -13979.978} C_VEL
LIN {X 0,Y 340.693,Z 163.545,A -85,B 0,C 180,E1 -13983.846,E2 -13983.846} C_VEL
LIN {X 0,Y 340.706,Z 163.545,A -85,B 0,C 180,E1 -13986.741,E2 -13986.741} C_VEL
LIN {X 0,Y 340.689,Z 163.549,A -85,B 0,C 180,E1 -13990.247,E2 -13990.247} C_VEL
LIN {X 0,Y 340.652,Z 163.551,A -85,B 0,C 180,E1 -13993.773,E2 -13993.773} C_VEL
LIN {X 0,Y 340.699,Z 163.547,A -85,B 0,C 180,E1 -13997.954,E2 -13997.954} C_VEL
LIN {X 0,Y 340.733,Z 163.542,A -85,B 0,C 180,E1 -14001.772,E2 -14001.772} C_VEL
LIN {X 0,Y 340.723,Z 163.543,A -85,B 0,C 180,E1 -14005.595,E2 -14005.595} C_VEL
LIN {X 0,Y 340.703,Z 163.543,A -85,B 0,C 180,E1 -14008.956,E2 -14008.956} C_VEL
LIN {X 0,Y 340.778,Z 163.532,A -85,B 0,C 180,E1 -14012.474,E2 -14012.474} C_VEL
LIN {X 0,Y 340.756,Z 163.54,A -85,B 0,C 180,E1 -14015.638,E2 -14015.638} C_VEL
LIN {X 0,Y 340.748,Z 163.542,A -85,B 0,C 180,E1 -14019.474,E2 -14019.474} C_VEL
LIN {X 0,Y 340.858,Z 163.524,A -85,B 0,C 180,E1 -14021.984,E2 -14021.984} C_VEL
LIN {X 0,Y 340.869,Z 163.523,A -85,B 0,C 180,E1 -14025.705,E2 -14025.705} C_VEL
LIN {X 0,Y 340.87,Z 163.525,A -85,B 0,C 180,E1 -14029.306,E2 -14029.306} C_VEL
LIN {X 0,Y 341.059,Z 163.501,A -85,B 0,C 180,E1 -14032.898,E2 -14032.898} C_VEL
LIN {X 0,Y 341.169,Z 163.483,A -85,B 0,C 180,E1 -14037.639,E2 -14037.639} C_VEL
LIN {X 0,Y 341.275,Z 163.47,A -85,B 0,C 180,E1 -14040,E2 -14040} C_VEL
LIN {X 0,Y 341.168,Z 163.487,A -85,B 0,C 180,E1 -14042.361,E2 -14042.361} C_VEL
LIN {X 0,Y 341.059,Z 163.499,A -85,B 0,C 180,E1 -14047.102,E2 -14047.102} C_VEL
LIN {X 0,Y 340.87,Z 163.525,A -85,B 0,C 180,E1 -14050.694,E2 -14050.694} C_VEL
LIN {X 0,Y 340.862,Z 163.526,A -85,B 0,C 180,E1 -14054.325,E2 -14054.325} C_VEL
LIN {X 0,Y 340.836,Z 163.527,A -85,B 0,C 180,E1 -14058.467,E2 -14058.467} C_VEL
LIN {X 0,Y 340.717,Z 163.543,A -85,B 0,C 180,E1 -14061.842,E2 -14061.842} C_VEL
LIN {X 0,Y 340.771,Z 163.535,A -85,B 0,C 180,E1 -14065.665,E2 -14065.665} C_VEL
LIN {X 0,Y 340.728,Z 163.542,A -85,B 0,C 180,E1 -14068.321,E2 -14068.321} C_VEL
LIN {X 0,Y 340.697,Z 163.543,A -85,B 0,C 180,E1 -14071.045,E2 -14071.045} C_VEL
LIN {X 0,Y 340.717,Z 163.542,A -85,B 0,C 180,E1 -14075.279,E2 -14075.279} C_VEL
LIN {X 0,Y 340.708,Z 163.542,A -85,B 0,C 180,E1 -14078.386,E2 -14078.386} C_VEL
LIN {X 0,Y 340.696,Z 163.545,A -85,B 0,C 180,E1 -14082.045,E2 -14082.045} C_VEL
LIN {X 0,Y 340.651,Z 163.549,A -85,B 0,C 180,E1 -14086.227,E2 -14086.227} C_VEL
LIN {X 0,Y 340.671,Z 163.547,A -85,B 0,C 180,E1 -14088.688,E2 -14088.688} C_VEL
LIN {X 0,Y 340.719,Z 163.542,A -85,B 0,C 180,E1 -14091.771,E2 -14091.771} C_VEL
LIN {X 0,Y 340.723,Z 163.543,A -85,B 0,C 180,E1 -14095.596,E2 -14095.596} C_VEL
LIN {X 0,Y 340.756,Z 163.67,A -85,B 0,C 180,E1 -14099.341,E2 -14099.341} C_VEL
LIN {X 0,Y 343.415,Z 176.125,A -85,B 0,C 180,E1 -14102.913,E2 -14102.913} C_VEL
LIN {X 0,Y 344.785,Z 183.655,A -85,B 0,C 180,E1 -14104.978,E2 -14104.978} C_VEL
LIN {X 0,Y 344.222,Z 189.742,A -85,B 0,C 180,E1 -14106.503,E2 -14106.503} C_VEL
LIN {X 0,Y 348.62,Z 213.948,A -85,B 0,C 180,E1 -14107.367,E2 -14107.367} C_VEL
LIN {X 0,Y 350.38,Z 226.187,A -85,B 0,C 180,E1 -14107.751,E2 -14107.751} C_VEL
LIN {X 0,Y 349.02,Z 298.198,A -85,B 0,C 180,E1 -14109.251,E2 -14109.251} C_VEL
LIN {X 0,Y 348.249,Z 311.385,A -85,B 0,C 180,E1 -14109.743,E2 -14109.743} C_VEL
LIN {X 0,Y 347.375,Z 323.502,A -85,B 0,C 180,E1 -14110.422,E2 -14110.422} C_VEL
LIN {X 0,Y 346.238,Z 335.732,A -85,B 0,C 180,E1 -14111.356,E2 -14111.356} C_VEL
LIN {X 0,Y 344.861,Z 347.305,A -85,B 0,C 180,E1 -14112.507,E2 -14112.507} C_VEL
LIN {X 0,Y 343.725,Z 357.212,A -85,B 0,C 180,E1 -14113.751,E2 -14113.751} C_VEL
LIN {X 0,Y 342.636,Z 366.255,A -85,B 0,C 180,E1 -14115.144,E2 -14115.144} C_VEL
LIN {X 0,Y 341.653,Z 374.12,A -85,B 0,C 180,E1 -14116.619,E2 -14116.619} C_VEL
LIN {X 0,Y 340.595,Z 381.799,A -85,B 0,C 180,E1 -14118.394,E2 -14118.394} C_VEL
LIN {X 0,Y 339.821,Z 388.886,A -85,B 0,C 180,E1 -14120.477,E2 -14120.477} C_VEL
LIN {X 0,Y 339.397,Z 393.601,A -85,B 0,C 180,E1 -14122.265,E2 -14122.265} C_VEL
LIN {X 0,Y 339.11,Z 397.38,A -85,B 0,C 180,E1 -14124.151,E2 -14124.151} C_VEL
LIN {X 0,Y 339.057,Z 399.062,A -85,B 0,C 180,E1 -14125.244,E2 -14125.244} C_VEL
LIN {X 0,Y 339.059,Z 400.457,A -85,B 0,C 180,E1 -14126.435,E2 -14126.435} C_VEL
LIN {X 0,Y 338.993,Z 402.057,A -85,B 0,C 180,E1 -14128.812,E2 -14128.812} C_VEL
LIN {X 0,Y 339.018,Z 402.271,A -85,B 0,C 180,E1 -14130,E2 -14130} C_VEL
LIN {X 0,Y 338.993,Z 402.051,A -85,B 0,C 180,E1 -14131.188,E2 -14131.188} C_VEL
LIN {X 0,Y 339.059,Z 400.444,A -85,B 0,C 180,E1 -14133.565,E2 -14133.565} C_VEL
LIN {X 0,Y 339.058,Z 399.044,A -85,B 0,C 180,E1 -14134.756,E2 -14134.756} C_VEL
LIN {X 0,Y 339.176,Z 396.104,A -85,B 0,C 180,E1 -14136.544,E2 -14136.544} C_VEL
LIN {X 0,Y 339.516,Z 392.128,A -85,B 0,C 180,E1 -14138.332,E2 -14138.332} C_VEL
LIN {X 0,Y 340.12,Z 386.014,A -85,B 0,C 180,E1 -14140.417,E2 -14140.417} C_VEL
LIN {X 0,Y 340.897,Z 379.337,A -85,B 0,C 180,E1 -14142.199,E2 -14142.199} C_VEL
LIN {X 0,Y 342.06,Z 371.058,A -85,B 0,C 180,E1 -14143.97,E2 -14143.97} C_VEL
LIN {X 0,Y 343.162,Z 361.427,A -85,B 0,C 180,E1 -14145.618,E2 -14145.618} C_VEL
LIN {X 0,Y 344.41,Z 350.894,A -85,B 0,C 180,E1 -14147.058,E2 -14147.058} C_VEL
LIN {X 0,Y 345.658,Z 340.262,A -85,B 0,C 180,E1 -14148.216,E2 -14148.216} C_VEL
LIN {X 0,Y 346.896,Z 328.374,A -85,B 0,C 180,E1 -14149.221,E2 -14149.221} C_VEL
LIN {X 0,Y 347.842,Z 317.302,A -85,B 0,C 180,E1 -14149.935,E2 -14149.935} C_VEL
LIN {X 0,Y 348.722,Z 304.194,A -85,B 0,C 180,E1 -14150.536,E2 -14150.536} C_VEL
LIN {X 0,Y 349.243,Z 291.648,A -85,B 0,C 180,E1 -14150.889,E2 -14150.889} C_VEL
LIN {X 0,Y 350.281,Z 224.93,A -85,B 0,C 180,E1 -14152.264,E2 -14152.264} C_VEL
LIN {X 0,Y 345.639,Z 197.202,A -85,B 0,C 180,E1 -14153.188,E2 -14153.188} C_VEL
LIN {X 0,Y 344.252,Z 189.684,A -85,B 0,C 180,E1 -14153.489,E2 -14153.489} C_VEL
LIN {X 0,Y 344.768,Z 183.574,A -85,B 0,C 180,E1 -14155.023,E2 -14155.023} C_VEL
LIN {X 0,Y 343.192,Z 174.786,A -85,B 0,C 180,E1 -14157.436,E2 -14157.436} C_VEL
LIN {X 0,Y 340.728,Z 163.538,A -85,B 0,C 180,E1 -14160.692,E2 -14160.692} C_VEL
LIN {X 0,Y 340.722,Z 163.542,A -85,B 0,C 180,E1 -14164.404,E2 -14164.404} C_VEL
LIN {X 0,Y 340.719,Z 163.543,A -85,B 0,C 180,E1 -14168.229,E2 -14168.229} C_VEL
LIN {X 0,Y 340.694,Z 163.545,A -85,B 0,C 180,E1 -14172.044,E2 -14172.044} C_VEL
LIN {X 0,Y 340.652,Z 163.552,A -85,B 0,C 180,E1 -14176.227,E2 -14176.227} C_VEL
LIN {X 0,Y 340.685,Z 163.546,A -85,B 0,C 180,E1 -14179.754,E2 -14179.754} C_VEL
LIN {X 0,Y 340.704,Z 163.543,A -85,B 0,C 180,E1 -14183.258,E2 -14183.258} C_VEL
LIN {X 0,Y 340.692,Z 163.549,A -85,B 0,C 180,E1 -14186.153,E2 -14186.153} C_VEL
LIN {X 0,Y 340.723,Z 163.545,A -85,B 0,C 180,E1 -14190.034,E2 -14190.034} C_VEL
LIN {X 0,Y 340.728,Z 163.538,A -85,B 0,C 180,E1 -14193.013,E2 -14193.013} C_VEL
LIN {X 0,Y 340.755,Z 163.539,A -85,B 0,C 180,E1 -14195.638,E2 -14195.638} C_VEL
LIN {X 0,Y 340.735,Z 163.541,A -85,B 0,C 180,E1 -14199.473,E2 -14199.473} C_VEL
LIN {X 0,Y 340.858,Z 163.526,A -85,B 0,C 180,E1 -14201.984,E2 -14201.984} C_VEL
LIN {X 0,Y 340.869,Z 163.527,A -85,B 0,C 180,E1 -14205.705,E2 -14205.705} C_VEL
LIN {X 0,Y 340.87,Z 163.524,A -85,B 0,C 180,E1 -14209.306,E2 -14209.306} C_VEL
LIN {X 0,Y 341.058,Z 163.499,A -85,B 0,C 180,E1 -14212.898,E2 -14212.898} C_VEL
LIN {X 0,Y 341.169,Z 163.486,A -85,B 0,C 180,E1 -14217.639,E2 -14217.639} C_VEL
LIN {X 0,Y 341.276,Z 163.47,A -85,B 0,C 180,E1 -14220,E2 -14220} C_VEL
LIN {X 0,Y 341.169,Z 163.485,A -85,B 0,C 180,E1 -14222.361,E2 -14222.361} C_VEL
LIN {X 0,Y 341.051,Z 163.504,A -85,B 0,C 180,E1 -14227.102,E2 -14227.102} C_VEL
LIN {X 0,Y 340.87,Z 163.525,A -85,B 0,C 180,E1 -14230.694,E2 -14230.694} C_VEL
LIN {X 0,Y 340.863,Z 163.524,A -85,B 0,C 180,E1 -14234.325,E2 -14234.325} C_VEL
LIN {X 0,Y 340.838,Z 163.528,A -85,B 0,C 180,E1 -14238.467,E2 -14238.467} C_VEL
LIN {X 0,Y 340.754,Z 163.536,A -85,B 0,C 180,E1 -14241.857,E2 -14241.857} C_VEL
LIN {X 0,Y 340.773,Z 163.534,A -85,B 0,C 180,E1 -14245.664,E2 -14245.664} C_VEL
LIN {X 0,Y 340.741,Z 163.542,A -85,B 0,C 180,E1 -14248.32,E2 -14248.32} C_VEL
LIN {X 0,Y 340.704,Z 163.542,A -85,B 0,C 180,E1 -14251.044,E2 -14251.044} C_VEL
LIN {X 0,Y 340.718,Z 163.54,A -85,B 0,C 180,E1 -14255.279,E2 -14255.279} C_VEL
LIN {X 0,Y 340.71,Z 163.544,A -85,B 0,C 180,E1 -14258.386,E2 -14258.386} C_VEL
LIN {X 0,Y 340.7,Z 163.548,A -85,B 0,C 180,E1 -14262.046,E2 -14262.046} C_VEL
LIN {X 0,Y 340.653,Z 163.551,A -85,B 0,C 180,E1 -14266.227,E2 -14266.227} C_VEL
LIN {X 0,Y 340.69,Z 163.549,A -85,B 0,C 180,E1 -14269.753,E2 -14269.753} C_VEL
LIN {X 0,Y 340.706,Z 163.545,A -85,B 0,C 180,E1 -14273.259,E2 -14273.259} C_VEL
LIN {X 0,Y 340.693,Z 163.545,A -85,B 0,C 180,E1 -14276.154,E2 -14276.154} C_VEL
LIN {X 0,Y 340.776,Z 163.536,A -85,B 0,C 180,E1 -14280.333,E2 -14280.333} C_VEL
LIN {X 0,Y 340.848,Z 163.696,A -85,B 0,C 180,E1 -14282.956,E2 -14282.956} C_VEL
LIN {X 0,Y 343.105,Z 174.556,A -85,B 0,C 180,E1 -14286.201,E2 -14286.201} C_VEL
LIN {X 0,Y 343.341,Z 175.92,A -85,B 0,C 180,E1 -14286.54,E2 -14286.54} C_VEL
LIN {X 0,Y 347.058,Z 186.275,A -85,B 0,C 180,E1 -14287.037,E2 -14287.037} C_VEL
LIN {X 0,Y 350.772,Z 205.493,A -85,B 0,C 180,E1 -14287.714,E2 -14287.714} C_VEL
LIN {X 0,Y 349.262,Z 282.509,A -85,B 0,C 180,E1 -14289.305,E2 -14289.305} C_VEL
LIN {X 0,Y 348.663,Z 295.185,A -85,B 0,C 180,E1 -14289.768,E2 -14289.768} C_VEL
LIN {X 0,Y 347.866,Z 307.6,A -85,B 0,C 180,E1 -14290.451,E2 -14290.451} C_VEL
LIN {X 0,Y 346.778,Z 320.075,A -85,B 0,C 180,E1 -14291.386,E2 -14291.386} C_VEL
LIN {X 0,Y 345.535,Z 331.99,A -85,B 0,C 180,E1 -14292.573,E2 -14292.573} C_VEL
LIN {X 0,Y 344.488,Z 342.13,A -85,B 0,C 180,E1 -14293.852,E2 -14293.852} C_VEL
LIN {X 0,Y 343.441,Z 350.74,A -85,B 0,C 180,E1 -14295.179,E2 -14295.179} C_VEL
LIN {X 0,Y 342.322,Z 358.616,A -85,B 0,C 180,E1 -14296.646,E2 -14296.646} C_VEL
LIN {X 0,Y 341.297,Z 366.312,A -85,B 0,C 180,E1 -14298.418,E2 -14298.418} C_VEL
LIN {X 0,Y 340.369,Z 373.376,A -85,B 0,C 180,E1 -14300.492,E2 -14300.492} C_VEL
LIN {X 0,Y 339.805,Z 378.08,A -85,B 0,C 180,E1 -14302.274,E2 -14302.274} C_VEL
LIN {X 0,Y 339.49,Z 381.679,A -85,B 0,C 180,E1 -14304.059,E2 -14304.059} C_VEL
LIN {X 0,Y 339.344,Z 383.538,A -85,B 0,C 180,E1 -14305.248,E2 -14305.248} C_VEL
LIN {X 0,Y 339.179,Z 384.939,A -85,B 0,C 180,E1 -14306.436,E2 -14306.436} C_VEL
LIN {X 0,Y 339.041,Z 386.548,A -85,B 0,C 180,E1 -14308.812,E2 -14308.812} C_VEL
LIN {X 0,Y 339.023,Z 386.781,A -85,B 0,C 180,E1 -14310,E2 -14310} C_VEL
LIN {X 0,Y 339.04,Z 386.59,A -85,B 0,C 180,E1 -14311.188,E2 -14311.188} C_VEL
LIN {X 0,Y 339.176,Z 385.036,A -85,B 0,C 180,E1 -14313.564,E2 -14313.564} C_VEL
LIN {X 0,Y 339.335,Z 383.678,A -85,B 0,C 180,E1 -14314.752,E2 -14314.752} C_VEL
LIN {X 0,Y 339.596,Z 380.695,A -85,B 0,C 180,E1 -14316.599,E2 -14316.599} C_VEL
LIN {X 0,Y 339.955,Z 376.919,A -85,B 0,C 180,E1 -14318.321,E2 -14318.321} C_VEL
LIN {X 0,Y 340.572,Z 371.898,A -85,B 0,C 180,E1 -14320.102,E2 -14320.102} C_VEL
LIN {X 0,Y 341.417,Z 365.576,A -85,B 0,C 180,E1 -14321.879,E2 -14321.879} C_VEL
LIN {X 0,Y 342.435,Z 357.664,A -85,B 0,C 180,E1 -14323.652,E2 -14323.652} C_VEL
LIN {X 0,Y 343.613,Z 349.595,A -85,B 0,C 180,E1 -14325.116,E2 -14325.116} C_VEL
LIN {X 0,Y 344.773,Z 339.274,A -85,B 0,C 180,E1 -14326.65,E2 -14326.65} C_VEL
LIN {X 0,Y 345.954,Z 328.677,A -85,B 0,C 180,E1 -14327.894,E2 -14327.894} C_VEL
LIN {X 0,Y 347.033,Z 317.817,A -85,B 0,C 180,E1 -14328.906,E2 -14328.906} C_VEL
LIN {X 0,Y 348.096,Z 305.816,A -85,B 0,C 180,E1 -14329.766,E2 -14329.766} C_VEL
LIN {X 0,Y 348.787,Z 293.507,A -85,B 0,C 180,E1 -14330.416,E2 -14330.416} C_VEL
LIN {X 0,Y 349.388,Z 280.784,A -85,B 0,C 180,E1 -14330.842,E2 -14330.842} C_VEL
LIN {X 0,Y 350.71,Z 209.572,A -85,B 0,C 180,E1 -14332.311,E2 -14332.311} C_VEL
LIN {X 0,Y 349.82,Z 203.856,A -85,B 0,C 180,E1 -14332.495,E2 -14332.495} C_VEL
LIN {X 0,Y 346.975,Z 196.776,A -85,B 0,C 180,E1 -14332.847,E2 -14332.847} C_VEL
LIN {X 0,Y 338.38,Z 181.66,A -85,B 0,C 180,E1 -14333.809,E2 -14333.809} C_VEL
LIN {X 0,Y 336.122,Z 175.77,A -85,B 0,C 180,E1 -14334.144,E2 -14334.144} C_VEL
LIN {X 0,Y 334.056,Z 165.642,A -85,B 0,C 180,E1 -14337.231,E2 -14337.231} C_VEL
LIN {X 0,Y 333.749,Z 164.411,A -85,B 0,C 180,E1 -14337.69,E2 -14337.69} C_VEL
LIN {X 0,Y 333.699,Z 164.42,A -85,B 0,C 180,E1 -14340.362,E2 -14340.362} C_VEL
LIN {X 0,Y 333.686,Z 164.42,A -85,B 0,C 180,E1 -14344.774,E2 -14344.774} C_VEL
LIN {X 0,Y 333.653,Z 164.421,A -85,B 0,C 180,E1 -14347.651,E2 -14347.651} C_VEL
LIN {X 0,Y 333.647,Z 164.424,A -85,B 0,C 180,E1 -14350.767,E2 -14350.767} C_VEL
LIN {X 0,Y 333.594,Z 164.432,A -85,B 0,C 180,E1 -14354.25,E2 -14354.25} C_VEL
LIN {X 0,Y 333.642,Z 164.424,A -85,B 0,C 180,E1 -14357.618,E2 -14357.618} C_VEL
LIN {X 0,Y 333.653,Z 164.421,A -85,B 0,C 180,E1 -14361.202,E2 -14361.202} C_VEL
LIN {X 0,Y 333.676,Z 164.422,A -85,B 0,C 180,E1 -14363.861,E2 -14363.861} C_VEL
LIN {X 0,Y 333.643,Z 164.422,A -85,B 0,C 180,E1 -14367.413,E2 -14367.413} C_VEL
LIN {X 0,Y 333.711,Z 164.413,A -85,B 0,C 180,E1 -14371.028,E2 -14371.028} C_VEL
LIN {X 0,Y 333.736,Z 164.415,A -85,B 0,C 180,E1 -14373.754,E2 -14373.754} C_VEL
LIN {X 0,Y 333.719,Z 164.412,A -85,B 0,C 180,E1 -14377.914,E2 -14377.914} C_VEL
LIN {X 0,Y 333.794,Z 164.407,A -85,B 0,C 180,E1 -14381.589,E2 -14381.589} C_VEL
LIN {X 0,Y 333.808,Z 164.404,A -85,B 0,C 180,E1 -14385.576,E2 -14385.576} C_VEL
LIN {X 0,Y 333.833,Z 164.404,A -85,B 0,C 180,E1 -14389.078,E2 -14389.078} C_VEL
LIN {X 0,Y 334.011,Z 164.376,A -85,B 0,C 180,E1 -14392.747,E2 -14392.747} C_VEL
LIN {X 0,Y 333.809,Z 164.405,A -85,B 0,C 180,E1 -14395.169,E2 -14395.169} C_VEL
LIN {X 0,Y 334.106,Z 164.363,A -85,B 0,C 180,E1 -14397.589,E2 -14397.589} C_VEL
LIN {X 0,Y 334.227,Z 164.348,A -85,B 0,C 180,E1 -14400,E2 -14400} C_VEL
LIN {X 0,Y 334.106,Z 164.367,A -85,B 0,C 180,E1 -14402.411,E2 -14402.411} C_VEL
LIN {X 0,Y 334.013,Z 164.374,A -85,B 0,C 180,E1 -14406.039,E2 -14406.039} C_VEL
LIN {X 0,Y 333.984,Z 164.384,A -85,B 0,C 180,E1 -14408.501,E2 -14408.501} C_VEL
LIN {X 0,Y 333.791,Z 164.406,A -85,B 0,C 180,E1 -14412.155,E2 -14412.155} C_VEL
LIN {X 0,Y 333.777,Z 164.407,A -85,B 0,C 180,E1 -14415.886,E2 -14415.886} C_VEL
LIN {X 0,Y 333.795,Z 164.402,A -85,B 0,C 180,E1 -14418.655,E2 -14418.655} C_VEL
LIN {X 0,Y 333.656,Z 164.425,A -85,B 0,C 180,E1 -14422.281,E2 -14422.281} C_VEL
LIN {X 0,Y 333.734,Z 164.414,A -85,B 0,C 180,E1 -14426.246,E2 -14426.246} C_VEL
LIN {X 0,Y 333.689,Z 164.416,A -85,B 0,C 180,E1 -14428.974,E2 -14428.974} C_VEL
LIN {X 0,Y 333.645,Z 164.422,A -85,B 0,C 180,E1 -14432.588,E2 -14432.588} C_VEL
LIN {X 0,Y 333.675,Z 164.42,A -85,B 0,C 180,E1 -14436.139,E2 -14436.139} C_VEL
LIN {X 0,Y 333.645,Z 164.423,A -85,B 0,C 180,E1 -14439.193,E2 -14439.193} C_VEL
LIN {X 0,Y 333.63,Z 164.424,A -85,B 0,C 180,E1 -14442.5,E2 -14442.5} C_VEL
LIN {X 0,Y 333.595,Z 164.429,A -85,B 0,C 180,E1 -14445.955,E2 -14445.955} C_VEL
LIN {X 0,Y 333.602,Z 164.432,A -85,B 0,C 180,E1 -14449.325,E2 -14449.325} C_VEL
LIN {X 0,Y 333.663,Z 164.424,A -85,B 0,C 180,E1 -14453.169,E2 -14453.169} C_VEL
LIN {X 0,Y 333.674,Z 164.423,A -85,B 0,C 180,E1 -14455.342,E2 -14455.342} C_VEL
LIN {X 0,Y 333.704,Z 164.621,A -85,B 0,C 180,E1 -14458.938,E2 -14458.938} C_VEL
LIN {X 0,Y 336.087,Z 175.353,A -85,B 0,C 180,E1 -14462.112,E2 -14462.112} C_VEL
LIN {X 0,Y 337.831,Z 184.733,A -85,B 0,C 180,E1 -14464.757,E2 -14464.757} C_VEL
LIN {X 0,Y 337.461,Z 189.669,A -85,B 0,C 180,E1 -14466.028,E2 -14466.028} C_VEL
LIN {X 0,Y 342.137,Z 215.189,A -85,B 0,C 180,E1 -14466.944,E2 -14466.944} C_VEL
LIN {X 0,Y 343.821,Z 226.612,A -85,B 0,C 180,E1 -14467.316,E2 -14467.316} C_VEL
LIN {X 0,Y 342.405,Z 298.05,A -85,B 0,C 180,E1 -14468.831,E2 -14468.831} C_VEL
LIN {X 0,Y 341.594,Z 311.231,A -85,B 0,C 180,E1 -14469.331,E2 -14469.331} C_VEL
LIN {X 0,Y 340.606,Z 324.461,A -85,B 0,C 180,E1 -14470.095,E2 -14470.095} C_VEL
LIN {X 0,Y 339.502,Z 335.574,A -85,B 0,C 180,E1 -14470.972,E2 -14470.972} C_VEL
LIN {X 0,Y 338.094,Z 347.147,A -85,B 0,C 180,E1 -14472.145,E2 -14472.145} C_VEL
LIN {X 0,Y 336.794,Z 357.882,A -85,B 0,C 180,E1 -14473.527,E2 -14473.527} C_VEL
LIN {X 0,Y 335.544,Z 367.768,A -85,B 0,C 180,E1 -14475.133,E2 -14475.133} C_VEL
LIN {X 0,Y 334.324,Z 376.693,A -85,B 0,C 180,E1 -14476.94,E2 -14476.94} C_VEL
LIN {X 0,Y 333.38,Z 383.875,A -85,B 0,C 180,E1 -14478.755,E2 -14478.755} C_VEL
LIN {X 0,Y 332.614,Z 390.418,A -85,B 0,C 180,E1 -14480.882,E2 -14480.882} C_VEL
LIN {X 0,Y 332.201,Z 394.748,A -85,B 0,C 180,E1 -14482.708,E2 -14482.708} C_VEL
LIN {X 0,Y 332.005,Z 397.546,A -85,B 0,C 180,E1 -14484.22,E2 -14484.22} C_VEL
LIN {X 0,Y 331.962,Z 400.295,A -85,B 0,C 180,E1 -14486.359,E2 -14486.359} C_VEL
LIN {X 0,Y 331.9,Z 401.895,A -85,B 0,C 180,E1 -14488.787,E2 -14488.787} C_VEL
LIN {X 0,Y 331.922,Z 402.109,A -85,B 0,C 180,E1 -14490,E2 -14490} C_VEL
LIN {X 0,Y 331.9,Z 401.889,A -85,B 0,C 180,E1 -14491.213,E2 -14491.213} C_VEL
LIN {X 0,Y 331.962,Z 400.282,A -85,B 0,C 180,E1 -14493.642,E2 -14493.642} C_VEL
LIN {X 0,Y 332.005,Z 397.521,A -85,B 0,C 180,E1 -14495.78,E2 -14495.78} C_VEL
LIN {X 0,Y 332.334,Z 393.397,A -85,B 0,C 180,E1 -14497.901,E2 -14497.901} C_VEL
LIN {X 0,Y 332.797,Z 388.671,A -85,B 0,C 180,E1 -14499.726,E2 -14499.726} C_VEL
LIN {X 0,Y 333.47,Z 382.693,A -85,B 0,C 180,E1 -14501.55,E2 -14501.55} C_VEL
LIN {X 0,Y 334.513,Z 375.253,A -85,B 0,C 180,E1 -14503.362,E2 -14503.362} C_VEL
LIN {X 0,Y 335.542,Z 367.67,A -85,B 0,C 180,E1 -14504.867,E2 -14504.867} C_VEL
LIN {X 0,Y 336.613,Z 358.881,A -85,B 0,C 180,E1 -14506.309,E2 -14506.309} C_VEL
LIN {X 0,Y 337.937,Z 348.283,A -85,B 0,C 180,E1 -14507.707,E2 -14507.707} C_VEL
LIN {X 0,Y 339.293,Z 336.964,A -85,B 0,C 180,E1 -14508.884,E2 -14508.884} C_VEL
LIN {X 0,Y 340.422,Z 325.218,A -85,B 0,C 180,E1 -14509.837,E2 -14509.837} C_VEL
LIN {X 0,Y 341.545,Z 312.366,A -85,B 0,C 180,E1 -14510.594,E2 -14510.594} C_VEL
LIN {X 0,Y 342.335,Z 299.757,A -85,B 0,C 180,E1 -14511.095,E2 -14511.095} C_VEL
LIN {X 0,Y 342.975,Z 275.356,A -85,B 0,C 180,E1 -14511.644,E2 -14511.644} C_VEL
LIN {X 0,Y 343.735,Z 225.833,A -85,B 0,C 180,E1 -14512.687,E2 -14512.687} C_VEL
LIN {X 0,Y 338.744,Z 196.134,A -85,B 0,C 180,E1 -14513.709,E2 -14513.709} C_VEL
LIN {X 0,Y 337.5,Z 189.552,A -85,B 0,C 180,E1 -14513.979,E2 -14513.979} C_VEL
LIN {X 0,Y 337.815,Z 184.65,A -85,B 0,C 180,E1 -14515.245,E2 -14515.245} C_VEL
LIN {X 0,Y 336.036,Z 175.27,A -85,B 0,C 180,E1 -14517.891,E2 -14517.891} C_VEL
LIN {X 0,Y 333.67,Z 164.419,A -85,B 0,C 180,E1 -14521.154,E2 -14521.154} C_VEL
LIN {X 0,Y 333.684,Z 164.422,A -85,B 0,C 180,E1 -14524.774,E2 -14524.774} C_VEL
LIN {X 0,Y 333.643,Z 164.423,A -85,B 0,C 180,E1 -14527.652,E2 -14527.652} C_VEL
LIN {X 0,Y 333.604,Z 164.433,A -85,B 0,C 180,E1 -14530.774,E2 -14530.774} C_VEL
LIN {X 0,Y 333.593,Z 164.432,A -85,B 0,C 180,E1 -14534.25,E2 -14534.25} C_VEL
LIN {X 0,Y 333.64,Z 164.423,A -85,B 0,C 180,E1 -14537.618,E2 -14537.618} C_VEL
LIN {X 0,Y 333.651,Z 164.421,A -85,B 0,C 180,E1 -14541.202,E2 -14541.202} C_VEL
LIN {X 0,Y 333.675,Z 164.42,A -85,B 0,C 180,E1 -14543.861,E2 -14543.861} C_VEL
LIN {X 0,Y 333.643,Z 164.422,A -85,B 0,C 180,E1 -14547.413,E2 -14547.413} C_VEL
LIN {X 0,Y 333.655,Z 164.421,A -85,B 0,C 180,E1 -14551.023,E2 -14551.023} C_VEL
LIN {X 0,Y 333.714,Z 164.413,A -85,B 0,C 180,E1 -14555.09,E2 -14555.09} C_VEL
LIN {X 0,Y 333.673,Z 164.418,A -85,B 0,C 180,E1 -14559.019,E2 -14559.019} C_VEL
LIN {X 0,Y 333.794,Z 164.407,A -85,B 0,C 180,E1 -14561.589,E2 -14561.589} C_VEL
LIN {X 0,Y 333.808,Z 164.407,A -85,B 0,C 180,E1 -14565.577,E2 -14565.577} C_VEL
LIN {X 0,Y 333.833,Z 164.399,A -85,B 0,C 180,E1 -14569.078,E2 -14569.078} C_VEL
LIN {X 0,Y 334.005,Z 164.376,A -85,B 0,C 180,E1 -14572.747,E2 -14572.747} C_VEL
LIN {X 0,Y 333.808,Z 164.404,A -85,B 0,C 180,E1 -14575.169,E2 -14575.169} C_VEL
LIN {X 0,Y 334.106,Z 164.367,A -85,B 0,C 180,E1 -14577.589,E2 -14577.589} C_VEL
LIN {X 0,Y 334.227,Z 164.348,A -85,B 0,C 180,E1 -14580,E2 -14580} C_VEL
LIN {X 0,Y 334.106,Z 164.365,A -85,B 0,C 180,E1 -14582.411,E2 -14582.411} C_VEL
LIN {X 0,Y 333.988,Z 164.377,A -85,B 0,C 180,E1 -14586.532,E2 -14586.532} C_VEL
LIN {X 0,Y 333.85,Z 164.396,A -85,B 0,C 180,E1 -14589.696,E2 -14589.696} C_VEL
LIN {X 0,Y 333.796,Z 164.404,A -85,B 0,C 180,E1 -14593.392,E2 -14593.392} C_VEL
LIN {X 0,Y 333.747,Z 164.409,A -85,B 0,C 180,E1 -14597.146,E2 -14597.146} C_VEL
LIN {X 0,Y 333.74,Z 164.41,A -85,B 0,C 180,E1 -14599.69,E2 -14599.69} C_VEL
LIN {X 0,Y 333.692,Z 164.418,A -85,B 0,C 180,E1 -14602.278,E2 -14602.278} C_VEL
LIN {X 0,Y 333.736,Z 164.414,A -85,B 0,C 180,E1 -14606.246,E2 -14606.246} C_VEL
LIN {X 0,Y 333.711,Z 164.414,A -85,B 0,C 180,E1 -14608.972,E2 -14608.972} C_VEL
LIN {X 0,Y 333.643,Z 164.425,A -85,B 0,C 180,E1 -14612.587,E2 -14612.587} C_VEL
LIN {X 0,Y 333.676,Z 164.422,A -85,B 0,C 180,E1 -14616.139,E2 -14616.139} C_VEL
LIN {X 0,Y 333.647,Z 164.421,A -85,B 0,C 180,E1 -14619.193,E2 -14619.193} C_VEL
LIN {X 0,Y 333.633,Z 164.424,A -85,B 0,C 180,E1 -14622.5,E2 -14622.5} C_VEL
LIN {X 0,Y 333.598,Z 164.433,A -85,B 0,C 180,E1 -14625.955,E2 -14625.955} C_VEL
LIN {X 0,Y 333.648,Z 164.423,A -85,B 0,C 180,E1 -14629.316,E2 -14629.316} C_VEL
LIN {X 0,Y 333.666,Z 164.422,A -85,B 0,C 180,E1 -14633.168,E2 -14633.168} C_VEL
LIN {X 0,Y 333.675,Z 164.423,A -85,B 0,C 180,E1 -14635.342,E2 -14635.342} C_VEL
LIN {X 0,Y 333.704,Z 164.419,A -85,B 0,C 180,E1 -14639.71,E2 -14639.71} C_VEL
LIN {X 0,Y 333.78,Z 164.529,A -85,B 0,C 180,E1 -14642.532,E2 -14642.532} C_VEL
LIN {X 0,Y 336.169,Z 175.816,A -85,B 0,C 180,E1 -14645.987,E2 -14645.987} C_VEL
LIN {X 0,Y 340.679,Z 188.125,A -85,B 0,C 180,E1 -14646.619,E2 -14646.619} C_VEL
LIN {X 0,Y 344.199,Z 206.216,A -85,B 0,C 180,E1 -14647.277,E2 -14647.277} C_VEL
LIN {X 0,Y 342.634,Z 282.689,A -85,B 0,C 180,E1 -14648.885,E2 -14648.885} C_VEL
LIN {X 0,Y 342.002,Z 296.117,A -85,B 0,C 180,E1 -14649.396,E2 -14649.396} C_VEL
LIN {X 0,Y 341.13,Z 308.897,A -85,B 0,C 180,E1 -14650.127,E2 -14650.127} C_VEL
LIN {X 0,Y 340.078,Z 320.243,A -85,B 0,C 180,E1 -14651.005,E2 -14651.005} C_VEL
LIN {X 0,Y 338.923,Z 330.74,A -85,B 0,C 180,E1 -14652.05,E2 -14652.05} C_VEL
LIN {X 0,Y 337.764,Z 341.225,A -85,B 0,C 180,E1 -14653.365,E2 -14653.365} C_VEL
LIN {X 0,Y 336.571,Z 350.905,A -85,B 0,C 180,E1 -14654.87,E2 -14654.87} C_VEL
LIN {X 0,Y 335.41,Z 358.781,A -85,B 0,C 180,E1 -14656.366,E2 -14656.366} C_VEL
LIN {X 0,Y 334.325,Z 366.477,A -85,B 0,C 180,E1 -14658.173,E2 -14658.173} C_VEL
LIN {X 0,Y 333.352,Z 373.54,A -85,B 0,C 180,E1 -14660.29,E2 -14660.29} C_VEL
LIN {X 0,Y 332.753,Z 378.244,A -85,B 0,C 180,E1 -14662.109,E2 -14662.109} C_VEL
LIN {X 0,Y 332.422,Z 381.842,A -85,B 0,C 180,E1 -14663.932,E2 -14663.932} C_VEL
LIN {X 0,Y 332.267,Z 383.701,A -85,B 0,C 180,E1 -14665.147,E2 -14665.147} C_VEL
LIN {X 0,Y 332.11,Z 385.101,A -85,B 0,C 180,E1 -14666.36,E2 -14666.36} C_VEL
LIN {X 0,Y 331.947,Z 386.71,A -85,B 0,C 180,E1 -14668.787,E2 -14668.787} C_VEL
LIN {X 0,Y 331.927,Z 386.943,A -85,B 0,C 180,E1 -14670,E2 -14670} C_VEL
LIN {X 0,Y 331.946,Z 386.752,A -85,B 0,C 180,E1 -14671.213,E2 -14671.213} C_VEL
LIN {X 0,Y 332.106,Z 385.198,A -85,B 0,C 180,E1 -14673.64,E2 -14673.64} C_VEL
LIN {X 0,Y 332.257,Z 383.839,A -85,B 0,C 180,E1 -14674.853,E2 -14674.853} C_VEL
LIN {X 0,Y 332.49,Z 381.183,A -85,B 0,C 180,E1 -14676.553,E2 -14676.553} C_VEL
LIN {X 0,Y 332.908,Z 377.08,A -85,B 0,C 180,E1 -14678.498,E2 -14678.498} C_VEL
LIN {X 0,Y 333.582,Z 372.059,A -85,B 0,C 180,E1 -14680.316,E2 -14680.316} C_VEL
LIN {X 0,Y 334.472,Z 365.736,A -85,B 0,C 180,E1 -14682.129,E2 -14682.129} C_VEL
LIN {X 0,Y 335.543,Z 357.824,A -85,B 0,C 180,E1 -14683.938,E2 -14683.938} C_VEL
LIN {X 0,Y 336.763,Z 349.754,A -85,B 0,C 180,E1 -14685.431,E2 -14685.431} C_VEL
LIN {X 0,Y 337.897,Z 339.912,A -85,B 0,C 180,E1 -14686.929,E2 -14686.929} C_VEL
LIN {X 0,Y 339.219,Z 328.834,A -85,B 0,C 180,E1 -14688.262,E2 -14688.262} C_VEL
LIN {X 0,Y 340.324,Z 317.973,A -85,B 0,C 180,E1 -14689.294,E2 -14689.294} C_VEL
LIN {X 0,Y 341.422,Z 305.971,A -85,B 0,C 180,E1 -14690.169,E2 -14690.169} C_VEL
LIN {X 0,Y 342.166,Z 293.657,A -85,B 0,C 180,E1 -14690.83,E2 -14690.83} C_VEL
LIN {X 0,Y 342.762,Z 280.925,A -85,B 0,C 180,E1 -14691.264,E2 -14691.264} C_VEL
LIN {X 0,Y 344.167,Z 206.527,A -85,B 0,C 180,E1 -14692.829,E2 -14692.829} C_VEL
LIN {X 0,Y 343.016,Z 199.294,A -85,B 0,C 180,E1 -14693.072,E2 -14693.072} C_VEL
LIN {X 0,Y 340.229,Z 186.571,A -85,B 0,C 180,E1 -14693.56,E2 -14693.56} C_VEL
LIN {X 0,Y 338.38,Z 181.66,A -85,B 0,C 180,E1 -14693.809,E2 -14693.809} C_VEL
LIN {X 0,Y 336.676,Z 178.675,A -85,B 0,C 180,E1 -14694.082,E2 -14694.082} C_VEL
LIN {X 0,Y 333.932,Z 175.183,A -85,B 0,C 180,E1 -14694.708,E2 -14694.708} C_VEL
LIN {X 0,Y 331.368,Z 172.501,A -85,B 0,C 180,E1 -14695.486,E2 -14695.486} C_VEL
LIN {X 0,Y 328.459,Z 169.221,A -85,B 0,C 180,E1 -14696.712,E2 -14696.712} C_VEL
LIN {X 0,Y 326.716,Z 165.494,A -85,B 0,C 180,E1 -14697.99,E2 -14697.99} C_VEL
LIN {X 0,Y 326.595,Z 165.304,A -85,B 0,C 180,E1 -14701.095,E2 -14701.095} C_VEL
LIN {X 0,Y 326.608,Z 165.301,A -85,B 0,C 180,E1 -14704.019,E2 -14704.019} C_VEL
LIN {X 0,Y 326.628,Z 165.296,A -85,B 0,C 180,E1 -14707.238,E2 -14707.238} C_VEL
LIN {X 0,Y 326.578,Z 165.303,A -85,B 0,C 180,E1 -14711.131,E2 -14711.131} C_VEL
LIN {X 0,Y 326.528,Z 165.309,A -85,B 0,C 180,E1 -14714.743,E2 -14714.743} C_VEL
LIN {X 0,Y 326.576,Z 165.306,A -85,B 0,C 180,E1 -14718.154,E2 -14718.154} C_VEL
LIN {X 0,Y 326.623,Z 165.297,A -85,B 0,C 180,E1 -14721.391,E2 -14721.391} C_VEL
LIN {X 0,Y 326.619,Z 165.297,A -85,B 0,C 180,E1 -14724.851,E2 -14724.851} C_VEL
LIN {X 0,Y 326.607,Z 165.298,A -85,B 0,C 180,E1 -14727.455,E2 -14727.455} C_VEL
LIN {X 0,Y 326.66,Z 165.292,A -85,B 0,C 180,E1 -14730.341,E2 -14730.341} C_VEL
LIN {X 0,Y 326.69,Z 165.288,A -85,B 0,C 180,E1 -14734.516,E2 -14734.516} C_VEL
LIN {X 0,Y 326.646,Z 165.291,A -85,B 0,C 180,E1 -14738.545,E2 -14738.545} C_VEL
LIN {X 0,Y 326.744,Z 165.285,A -85,B 0,C 180,E1 -14741.177,E2 -14741.177} C_VEL
LIN {X 0,Y 326.763,Z 165.282,A -85,B 0,C 180,E1 -14745.433,E2 -14745.433} C_VEL
LIN {X 0,Y 326.769,Z 165.281,A -85,B 0,C 180,E1 -14748.839,E2 -14748.839} C_VEL
LIN {X 0,Y 326.965,Z 165.252,A -85,B 0,C 180,E1 -14752.59,E2 -14752.59} C_VEL
LIN {X 0,Y 326.775,Z 165.282,A -85,B 0,C 180,E1 -14755.065,E2 -14755.065} C_VEL
LIN {X 0,Y 327.047,Z 165.242,A -85,B 0,C 180,E1 -14757.537,E2 -14757.537} C_VEL
LIN {X 0,Y 327.179,Z 165.225,A -85,B 0,C 180,E1 -14760,E2 -14760} C_VEL
LIN {X 0,Y 327.046,Z 165.247,A -85,B 0,C 180,E1 -14762.463,E2 -14762.463} C_VEL
LIN {X 0,Y 326.989,Z 165.249,A -85,B 0,C 180,E1 -14766.169,E2 -14766.169} C_VEL
LIN {X 0,Y 326.914,Z 165.265,A -85,B 0,C 180,E1 -14768.655,E2 -14768.655} C_VEL
LIN {X 0,Y 326.734,Z 165.284,A -85,B 0,C 180,E1 -14772.421,E2 -14772.421} C_VEL
LIN {X 0,Y 326.753,Z 165.281,A -85,B 0,C 180,E1 -14774.958,E2 -14774.958} C_VEL
LIN {X 0,Y 326.732,Z 165.281,A -85,B 0,C 180,E1 -14778.838,E2 -14778.838} C_VEL
LIN {X 0,Y 326.602,Z 165.3,A -85,B 0,C 180,E1 -14782.789,E2 -14782.789} C_VEL
LIN {X 0,Y 326.689,Z 165.287,A -85,B 0,C 180,E1 -14785.484,E2 -14785.484} C_VEL
LIN {X 0,Y 326.647,Z 165.297,A -85,B 0,C 180,E1 -14789.66,E2 -14789.66} C_VEL
LIN {X 0,Y 326.618,Z 165.298,A -85,B 0,C 180,E1 -14792.947,E2 -14792.947} C_VEL
LIN {X 0,Y 326.612,Z 165.3,A -85,B 0,C 180,E1 -14795.52,E2 -14795.52} C_VEL
LIN {X 0,Y 326.61,Z 165.299,A -85,B 0,C 180,E1 -14799.227,E2 -14799.227} C_VEL
LIN {X 0,Y 326.574,Z 165.304,A -85,B 0,C 180,E1 -14802.972,E2 -14802.972} C_VEL
LIN {X 0,Y 326.573,Z 165.305,A -85,B 0,C 180,E1 -14807.029,E2 -14807.029} C_VEL
LIN {X 0,Y 326.582,Z 165.306,A -85,B 0,C 180,E1 -14811.386,E2 -14811.386} C_VEL
LIN {X 0,Y 326.619,Z 165.301,A -85,B 0,C 180,E1 -14814.852,E2 -14814.852} C_VEL
LIN {X 0,Y 326.614,Z 165.38,A -85,B 0,C 180,E1 -14818.456,E2 -14818.456} C_VEL
LIN {X 0,Y 329.224,Z 177.025,A -85,B 0,C 180,E1 -14821.989,E2 -14821.989} C_VEL
LIN {X 0,Y 330.971,Z 187.06,A -85,B 0,C 180,E1 -14824.869,E2 -14824.869} C_VEL
LIN {X 0,Y 330.748,Z 189.452,A -85,B 0,C 180,E1 -14825.496,E2 -14825.496} C_VEL
LIN {X 0,Y 335.688,Z 216.618,A -85,B 0,C 180,E1 -14826.51,E2 -14826.51} C_VEL
LIN {X 0,Y 337.288,Z 227.274,A -85,B 0,C 180,E1 -14826.869,E2 -14826.869} C_VEL
LIN {X 0,Y 335.805,Z 297.901,A -85,B 0,C 180,E1 -14828.394,E2 -14828.394} C_VEL
LIN {X 0,Y 334.97,Z 311.078,A -85,B 0,C 180,E1 -14828.903,E2 -14828.903} C_VEL
LIN {X 0,Y 333.937,Z 324.305,A -85,B 0,C 180,E1 -14829.68,E2 -14829.68} C_VEL
LIN {X 0,Y 332.784,Z 335.416,A -85,B 0,C 180,E1 -14830.572,E2 -14830.572} C_VEL
LIN {X 0,Y 331.34,Z 346.988,A -85,B 0,C 180,E1 -14831.768,E2 -14831.768} C_VEL
LIN {X 0,Y 329.965,Z 357.732,A -85,B 0,C 180,E1 -14833.178,E2 -14833.178} C_VEL
LIN {X 0,Y 328.647,Z 367.607,A -85,B 0,C 180,E1 -14834.814,E2 -14834.814} C_VEL
LIN {X 0,Y 327.377,Z 376.532,A -85,B 0,C 180,E1 -14836.657,E2 -14836.657} C_VEL
LIN {X 0,Y 326.371,Z 383.713,A -85,B 0,C 180,E1 -14838.511,E2 -14838.511} C_VEL
LIN {X 0,Y 325.583,Z 390.256,A -85,B 0,C 180,E1 -14840.683,E2 -14840.683} C_VEL
LIN {X 0,Y 325.152,Z 394.587,A -85,B 0,C 180,E1 -14842.549,E2 -14842.549} C_VEL
LIN {X 0,Y 324.908,Z 397.652,A -85,B 0,C 180,E1 -14844.278,E2 -14844.278} C_VEL
LIN {X 0,Y 324.869,Z 400.133,A -85,B 0,C 180,E1 -14846.279,E2 -14846.279} C_VEL
LIN {X 0,Y 324.829,Z 401.127,A -85,B 0,C 180,E1 -14847.52,E2 -14847.52} C_VEL
LIN {X 0,Y 324.81,Z 401.733,A -85,B 0,C 180,E1 -14848.76,E2 -14848.76} C_VEL
LIN {X 0,Y 324.829,Z 401.947,A -85,B 0,C 180,E1 -14850,E2 -14850} C_VEL
LIN {X 0,Y 324.81,Z 401.727,A -85,B 0,C 180,E1 -14851.24,E2 -14851.24} C_VEL
LIN {X 0,Y 324.829,Z 401.117,A -85,B 0,C 180,E1 -14852.48,E2 -14852.48} C_VEL
LIN {X 0,Y 324.869,Z 400.119,A -85,B 0,C 180,E1 -14853.721,E2 -14853.721} C_VEL
LIN {X 0,Y 324.908,Z 397.627,A -85,B 0,C 180,E1 -14855.723,E2 -14855.723} C_VEL
LIN {X 0,Y 325.152,Z 394.549,A -85,B 0,C 180,E1 -14857.452,E2 -14857.452} C_VEL
LIN {X 0,Y 325.583,Z 390.205,A -85,B 0,C 180,E1 -14859.317,E2 -14859.317} C_VEL
LIN {X 0,Y 326.247,Z 384.674,A -85,B 0,C 180,E1 -14861.179,E2 -14861.179} C_VEL
LIN {X 0,Y 327.198,Z 377.773,A -85,B 0,C 180,E1 -14863.034,E2 -14863.034} C_VEL
LIN {X 0,Y 328.415,Z 369.137,A -85,B 0,C 180,E1 -14864.88,E2 -14864.88} C_VEL
LIN {X 0,Y 329.522,Z 360.478,A -85,B 0,C 180,E1 -14866.383,E2 -14866.383} C_VEL
LIN {X 0,Y 330.829,Z 350.562,A -85,B 0,C 180,E1 -14867.781,E2 -14867.781} C_VEL
LIN {X 0,Y 332.19,Z 339.929,A -85,B 0,C 180,E1 -14868.983,E2 -14868.983} C_VEL
LIN {X 0,Y 333.475,Z 328.037,A -85,B 0,C 180,E1 -14870.027,E2 -14870.027} C_VEL
LIN {X 0,Y 334.544,Z 316.963,A -85,B 0,C 180,E1 -14870.763,E2 -14870.763} C_VEL
LIN {X 0,Y 335.434,Z 304.764,A -85,B 0,C 180,E1 -14871.349,E2 -14871.349} C_VEL
LIN {X 0,Y 336.036,Z 291.283,A -85,B 0,C 180,E1 -14871.751,E2 -14871.751} C_VEL
LIN {X 0,Y 337.103,Z 226.177,A -85,B 0,C 180,E1 -14873.147,E2 -14873.147} C_VEL
LIN {X 0,Y 332.38,Z 198.001,A -85,B 0,C 180,E1 -14874.144,E2 -14874.144} C_VEL
LIN {X 0,Y 330.702,Z 189.46,A -85,B 0,C 180,E1 -14874.483,E2 -14874.483} C_VEL
LIN {X 0,Y 330.85,Z 185.723,A -85,B 0,C 180,E1 -14875.477,E2 -14875.477} C_VEL
LIN {X 0,Y 328.8,Z 175.267,A -85,B 0,C 180,E1 -14878.51,E2 -14878.51} C_VEL
LIN {X 0,Y 326.612,Z 165.297,A -85,B 0,C 180,E1 -14881.544,E2 -14881.544} C_VEL
LIN {X 0,Y 326.611,Z 165.3,A -85,B 0,C 180,E1 -14885.52,E2 -14885.52} C_VEL
LIN {X 0,Y 326.588,Z 165.304,A -85,B 0,C 180,E1 -14889.222,E2 -14889.222} C_VEL
LIN {X 0,Y 326.574,Z 165.306,A -85,B 0,C 180,E1 -14892.971,E2 -14892.971} C_VEL
LIN {X 0,Y 326.575,Z 165.304,A -85,B 0,C 180,E1 -14897.028,E2 -14897.028} C_VEL
LIN {X 0,Y 326.61,Z 165.301,A -85,B 0,C 180,E1 -14900.773,E2 -14900.773} C_VEL
LIN {X 0,Y 326.612,Z 165.302,A -85,B 0,C 180,E1 -14904.48,E2 -14904.48} C_VEL
LIN {X 0,Y 326.608,Z 165.299,A -85,B 0,C 180,E1 -14907.455,E2 -14907.455} C_VEL
LIN {X 0,Y 326.617,Z 165.301,A -85,B 0,C 180,E1 -14910.337,E2 -14910.337} C_VEL
LIN {X 0,Y 326.62,Z 165.296,A -85,B 0,C 180,E1 -14913.137,E2 -14913.137} C_VEL
LIN {X 0,Y 326.643,Z 165.299,A -85,B 0,C 180,E1 -14915.87,E2 -14915.87} C_VEL
LIN {X 0,Y 326.658,Z 165.297,A -85,B 0,C 180,E1 -14919.865,E2 -14919.865} C_VEL
LIN {X 0,Y 326.699,Z 165.286,A -85,B 0,C 180,E1 -14922.472,E2 -14922.472} C_VEL
LIN {X 0,Y 326.759,Z 165.279,A -85,B 0,C 180,E1 -14926.315,E2 -14926.315} C_VEL
LIN {X 0,Y 326.805,Z 165.275,A -85,B 0,C 180,E1 -14930.094,E2 -14930.094} C_VEL
LIN {X 0,Y 326.988,Z 165.252,A -85,B 0,C 180,E1 -14933.831,E2 -14933.831} C_VEL
LIN {X 0,Y 327.047,Z 165.246,A -85,B 0,C 180,E1 -14937.537,E2 -14937.537} C_VEL
LIN {X 0,Y 327.179,Z 165.226,A -85,B 0,C 180,E1 -14940,E2 -14940} C_VEL
LIN {X 0,Y 327.047,Z 165.244,A -85,B 0,C 180,E1 -14942.463,E2 -14942.463} C_VEL
LIN {X 0,Y 326.96,Z 165.252,A -85,B 0,C 180,E1 -14946.523,E2 -14946.523} C_VEL
LIN {X 0,Y 326.805,Z 165.273,A -85,B 0,C 180,E1 -14949.907,E2 -14949.907} C_VEL
LIN {X 0,Y 326.759,Z 165.28,A -85,B 0,C 180,E1 -14953.685,E2 -14953.685} C_VEL
LIN {X 0,Y 326.699,Z 165.285,A -85,B 0,C 180,E1 -14957.528,E2 -14957.528} C_VEL
LIN {X 0,Y 326.665,Z 165.293,A -85,B 0,C 180,E1 -14960.135,E2 -14960.135} C_VEL
LIN {X 0,Y 326.652,Z 165.294,A -85,B 0,C 180,E1 -14964.129,E2 -14964.129} C_VEL
LIN {X 0,Y 326.685,Z 165.289,A -85,B 0,C 180,E1 -14966.858,E2 -14966.858} C_VEL
LIN {X 0,Y 326.639,Z 165.297,A -85,B 0,C 180,E1 -14970.611,E2 -14970.611} C_VEL
LIN {X 0,Y 326.607,Z 165.302,A -85,B 0,C 180,E1 -14974.02,E2 -14974.02} C_VEL
LIN {X 0,Y 326.628,Z 165.296,A -85,B 0,C 180,E1 -14977.239,E2 -14977.239} C_VEL
LIN {X 0,Y 326.578,Z 165.303,A -85,B 0,C 180,E1 -14981.132,E2 -14981.132} C_VEL
LIN {X 0,Y 326.528,Z 165.308,A -85,B 0,C 180,E1 -14984.743,E2 -14984.743} C_VEL
LIN {X 0,Y 326.577,Z 165.305,A -85,B 0,C 180,E1 -14988.155,E2 -14988.155} C_VEL
LIN {X 0,Y 326.624,Z 165.3,A -85,B 0,C 180,E1 -14991.392,E2 -14991.392} C_VEL
LIN {X 0,Y 326.62,Z 165.299,A -85,B 0,C 180,E1 -14994.852,E2 -14994.852} C_VEL
LIN {X 0,Y 326.609,Z 165.302,A -85,B 0,C 180,E1 -14997.456,E2 -14997.456} C_VEL
LIN {X 0,Y 326.662,Z 165.295,A -85,B 0,C 180,E1 -15000.341,E2 -15000.341} C_VEL
LIN {X 0,Y 326.698,Z 165.399,A -85,B 0,C 180,E1 -15002.096,E2 -15002.096} C_VEL
LIN {X 0,Y 328.803,Z 175.121,A -85,B 0,C 180,E1 -15005.161,E2 -15005.161} C_VEL
LIN {X 0,Y 328.978,Z 175.997,A -85,B 0,C 180,E1 -15005.429,E2 -15005.429} C_VEL
LIN {X 0,Y 334.494,Z 190.699,A -85,B 0,C 180,E1 -15006.216,E2 -15006.216} C_VEL
LIN {X 0,Y 337.649,Z 206.768,A -85,B 0,C 180,E1 -15006.819,E2 -15006.819} C_VEL
LIN {X 0,Y 336.128,Z 281.419,A -85,B 0,C 180,E1 -15008.416,E2 -15008.416} C_VEL
LIN {X 0,Y 335.496,Z 293.992,A -85,B 0,C 180,E1 -15008.857,E2 -15008.857} C_VEL
LIN {X 0,Y 334.638,Z 306.811,A -85,B 0,C 180,E1 -15009.564,E2 -15009.564} C_VEL
LIN {X 0,Y 333.545,Z 318.67,A -85,B 0,C 180,E1 -15010.458,E2 -15010.458} C_VEL
LIN {X 0,Y 332.371,Z 329.429,A -85,B 0,C 180,E1 -15011.508,E2 -15011.508} C_VEL
LIN {X 0,Y 331.133,Z 339.655,A -85,B 0,C 180,E1 -15012.763,E2 -15012.763} C_VEL
LIN {X 0,Y 330.011,Z 349.294,A -85,B 0,C 180,E1 -15014.245,E2 -15014.245} C_VEL
LIN {X 0,Y 328.511,Z 358.946,A -85,B 0,C 180,E1 -15016.074,E2 -15016.074} C_VEL
LIN {X 0,Y 327.376,Z 366.641,A -85,B 0,C 180,E1 -15017.918,E2 -15017.918} C_VEL
LIN {X 0,Y 326.354,Z 373.704,A -85,B 0,C 180,E1 -15020.08,E2 -15020.08} C_VEL
LIN {X 0,Y 325.726,Z 378.407,A -85,B 0,C 180,E1 -15021.938,E2 -15021.938} C_VEL
LIN {X 0,Y 325.37,Z 382.005,A -85,B 0,C 180,E1 -15023.8,E2 -15023.8} C_VEL
LIN {X 0,Y 325.193,Z 383.864,A -85,B 0,C 180,E1 -15025.041,E2 -15025.041} C_VEL
LIN {X 0,Y 325.042,Z 385.264,A -85,B 0,C 180,E1 -15026.281,E2 -15026.281} C_VEL
LIN {X 0,Y 324.856,Z 386.872,A -85,B 0,C 180,E1 -15028.76,E2 -15028.76} C_VEL
LIN {X 0,Y 324.834,Z 387.105,A -85,B 0,C 180,E1 -15030,E2 -15030} C_VEL
LIN {X 0,Y 324.855,Z 386.914,A -85,B 0,C 180,E1 -15031.24,E2 -15031.24} C_VEL
LIN {X 0,Y 325.038,Z 385.359,A -85,B 0,C 180,E1 -15033.719,E2 -15033.719} C_VEL
LIN {X 0,Y 325.183,Z 384.001,A -85,B 0,C 180,E1 -15034.959,E2 -15034.959} C_VEL
LIN {X 0,Y 325.382,Z 381.677,A -85,B 0,C 180,E1 -15036.501,E2 -15036.501} C_VEL
LIN {X 0,Y 325.879,Z 377.241,A -85,B 0,C 180,E1 -15038.683,E2 -15038.683} C_VEL
LIN {X 0,Y 326.604,Z 372.219,A -85,B 0,C 180,E1 -15040.539,E2 -15040.539} C_VEL
LIN {X 0,Y 327.535,Z 365.897,A -85,B 0,C 180,E1 -15042.39,E2 -15042.39} C_VEL
LIN {X 0,Y 328.664,Z 357.983,A -85,B 0,C 180,E1 -15044.236,E2 -15044.236} C_VEL
LIN {X 0,Y 329.92,Z 349.913,A -85,B 0,C 180,E1 -15045.759,E2 -15045.759} C_VEL
LIN {X 0,Y 331.123,Z 340.07,A -85,B 0,C 180,E1 -15047.286,E2 -15047.286} C_VEL
LIN {X 0,Y 332.48,Z 328.991,A -85,B 0,C 180,E1 -15048.645,E2 -15048.645} C_VEL
LIN {X 0,Y 333.643,Z 318.129,A -85,B 0,C 180,E1 -15049.696,E2 -15049.696} C_VEL
LIN {X 0,Y 334.781,Z 306.125,A -85,B 0,C 180,E1 -15050.587,E2 -15050.587} C_VEL
LIN {X 0,Y 335.553,Z 293.807,A -85,B 0,C 180,E1 -15051.26,E2 -15051.26} C_VEL
LIN {X 0,Y 336.173,Z 281.066,A -85,B 0,C 180,E1 -15051.701,E2 -15051.701} C_VEL
LIN {X 0,Y 337.558,Z 205.866,A -85,B 0,C 180,E1 -15053.32,E2 -15053.32} C_VEL
LIN {X 0,Y 334.173,Z 189.449,A -85,B 0,C 180,E1 -15053.95,E2 -15053.95} C_VEL
LIN {X 0,Y 328.982,Z 176.01,A -85,B 0,C 180,E1 -15054.682,E2 -15054.682} C_VEL
LIN {X 0,Y 327.066,Z 166.965,A -85,B 0,C 180,E1 -15057.516,E2 -15057.516} C_VEL
LIN {X 0,Y 326.716,Z 165.494,A -85,B 0,C 180,E1 -15057.99,E2 -15057.99} C_VEL
LIN {X 0,Y 326.015,Z 165.377,A -85,B 0,C 180,E1 -15058.616,E2 -15058.616} C_VEL
LIN {X 0,Y 322.698,Z 165.791,A -85,B 0,C 180,E1 -15060.607,E2 -15060.607} C_VEL
LIN {X 0,Y 320.569,Z 166.273,A -85,B 0,C 180,E1 -15062.006,E2 -15062.006} C_VEL
LIN {X 0,Y 319.569,Z 166.176,A -85,B 0,C 180,E1 -15063.452,E2 -15063.452} C_VEL
LIN {X 0,Y 319.559,Z 166.182,A -85,B 0,C 180,E1 -15066.427,E2 -15066.427} C_VEL
LIN {X 0,Y 319.559,Z 166.177,A -85,B 0,C 180,E1 -15069.668,E2 -15069.668} C_VEL
LIN {X 0,Y 319.522,Z 166.182,A -85,B 0,C 180,E1 -15073.46,E2 -15073.46} C_VEL
LIN {X 0,Y 319.554,Z 166.177,A -85,B 0,C 180,E1 -15077.016,E2 -15077.016} C_VEL
LIN {X 0,Y 319.547,Z 166.18,A -85,B 0,C 180,E1 -15080.371,E2 -15080.371} C_VEL
LIN {X 0,Y 319.558,Z 166.178,A -85,B 0,C 180,E1 -15083.572,E2 -15083.572} C_VEL
LIN {X 0,Y 319.577,Z 166.171,A -85,B 0,C 180,E1 -15086.686,E2 -15086.686} C_VEL
LIN {X 0,Y 319.591,Z 166.177,A -85,B 0,C 180,E1 -15089.616,E2 -15089.616} C_VEL
LIN {X 0,Y 319.608,Z 166.168,A -85,B 0,C 180,E1 -15092.498,E2 -15092.498} C_VEL
LIN {X 0,Y 319.605,Z 166.174,A -85,B 0,C 180,E1 -15095.304,E2 -15095.304} C_VEL
LIN {X 0,Y 319.597,Z 166.17,A -85,B 0,C 180,E1 -15098.048,E2 -15098.048} C_VEL
LIN {X 0,Y 319.689,Z 166.162,A -85,B 0,C 180,E1 -15100.962,E2 -15100.962} C_VEL
LIN {X 0,Y 319.73,Z 166.156,A -85,B 0,C 180,E1 -15105.276,E2 -15105.276} C_VEL
LIN {X 0,Y 319.756,Z 166.15,A -85,B 0,C 180,E1 -15109.873,E2 -15109.873} C_VEL
LIN {X 0,Y 319.924,Z 166.128,A -85,B 0,C 180,E1 -15112.426,E2 -15112.426} C_VEL
LIN {X 0,Y 319.745,Z 166.159,A -85,B 0,C 180,E1 -15114.956,E2 -15114.956} C_VEL
LIN {X 0,Y 319.99,Z 166.121,A -85,B 0,C 180,E1 -15117.482,E2 -15117.482} C_VEL
LIN {X 0,Y 320.131,Z 166.103,A -85,B 0,C 180,E1 -15120,E2 -15120} C_VEL
LIN {X 0,Y 319.99,Z 166.126,A -85,B 0,C 180,E1 -15122.518,E2 -15122.518} C_VEL
LIN {X 0,Y 319.944,Z 166.127,A -85,B 0,C 180,E1 -15126.306,E2 -15126.306} C_VEL
LIN {X 0,Y 319.842,Z 166.144,A -85,B 0,C 180,E1 -15128.848,E2 -15128.848} C_VEL
LIN {X 0,Y 319.681,Z 166.16,A -85,B 0,C 180,E1 -15132.7,E2 -15132.7} C_VEL
LIN {X 0,Y 319.699,Z 166.158,A -85,B 0,C 180,E1 -15135.296,E2 -15135.296} C_VEL
LIN {X 0,Y 319.651,Z 166.161,A -85,B 0,C 180,E1 -15139.256,E2 -15139.256} C_VEL
LIN {X 0,Y 319.559,Z 166.177,A -85,B 0,C 180,E1 -15143.32,E2 -15143.32} C_VEL
LIN {X 0,Y 319.633,Z 166.17,A -85,B 0,C 180,E1 -15146.088,E2 -15146.088} C_VEL
LIN {X 0,Y 319.579,Z 166.174,A -85,B 0,C 180,E1 -15148.935,E2 -15148.935} C_VEL
LIN {X 0,Y 319.531,Z 166.185,A -85,B 0,C 180,E1 -15151.862,E2 -15151.862} C_VEL
LIN {X 0,Y 319.579,Z 166.176,A -85,B 0,C 180,E1 -15155.543,E2 -15155.543} C_VEL
LIN {X 0,Y 319.558,Z 166.182,A -85,B 0,C 180,E1 -15159.669,E2 -15159.669} C_VEL
LIN {X 0,Y 319.52,Z 166.186,A -85,B 0,C 180,E1 -15163.461,E2 -15163.461} C_VEL
LIN {X 0,Y 319.552,Z 166.18,A -85,B 0,C 180,E1 -15167.016,E2 -15167.016} C_VEL
LIN {X 0,Y 319.544,Z 166.179,A -85,B 0,C 180,E1 -15170.371,E2 -15170.371} C_VEL
LIN {X 0,Y 319.58,Z 166.176,A -85,B 0,C 180,E1 -15174.457,E2 -15174.457} C_VEL
LIN {X 0,Y 319.601,Z 166.298,A -85,B 0,C 180,E1 -15178.007,E2 -15178.007} C_VEL
LIN {X 0,Y 321.93,Z 176.843,A -85,B 0,C 180,E1 -15181.297,E2 -15181.297} C_VEL
LIN {X 0,Y 323.883,Z 186.885,A -85,B 0,C 180,E1 -15184.28,E2 -15184.28} C_VEL
LIN {X 0,Y 324.01,Z 189.273,A -85,B 0,C 180,E1 -15184.948,E2 -15184.948} C_VEL
LIN {X 0,Y 329.182,Z 217.597,A -85,B 0,C 180,E1 -15186.044,E2 -15186.044} C_VEL
LIN {X 0,Y 330.758,Z 229.119,A -85,B 0,C 180,E1 -15186.431,E2 -15186.431} C_VEL
LIN {X 0,Y 329.223,Z 297.752,A -85,B 0,C 180,E1 -15187.94,E2 -15187.94} C_VEL
LIN {X 0,Y 328.363,Z 310.925,A -85,B 0,C 180,E1 -15188.457,E2 -15188.457} C_VEL
LIN {X 0,Y 327.274,Z 324.149,A -85,B 0,C 180,E1 -15189.248,E2 -15189.248} C_VEL
LIN {X 0,Y 326.08,Z 335.258,A -85,B 0,C 180,E1 -15190.156,E2 -15190.156} C_VEL
LIN {X 0,Y 324.584,Z 346.829,A -85,B 0,C 180,E1 -15191.375,E2 -15191.375} C_VEL
LIN {X 0,Y 323.14,Z 357.573,A -85,B 0,C 180,E1 -15192.812,E2 -15192.812} C_VEL
LIN {X 0,Y 321.99,Z 366.118,A -85,B 0,C 180,E1 -15194.23,E2 -15194.23} C_VEL
LIN {X 0,Y 320.693,Z 375.013,A -85,B 0,C 180,E1 -15196.051,E2 -15196.051} C_VEL
LIN {X 0,Y 319.514,Z 382.436,A -85,B 0,C 180,E1 -15197.939,E2 -15197.939} C_VEL
LIN {X 0,Y 318.759,Z 388.402,A -85,B 0,C 180,E1 -15199.841,E2 -15199.841} C_VEL
LIN {X 0,Y 318.213,Z 393.116,A -85,B 0,C 180,E1 -15201.746,E2 -15201.746} C_VEL
LIN {X 0,Y 317.89,Z 396.718,A -85,B 0,C 180,E1 -15203.654,E2 -15203.654} C_VEL
LIN {X 0,Y 317.791,Z 398.576,A -85,B 0,C 180,E1 -15204.925,E2 -15204.925} C_VEL
LIN {X 0,Y 317.778,Z 399.971,A -85,B 0,C 180,E1 -15206.196,E2 -15206.196} C_VEL
LIN {X 0,Y 317.75,Z 400.965,A -85,B 0,C 180,E1 -15207.465,E2 -15207.465} C_VEL
LIN {X 0,Y 317.722,Z 401.571,A -85,B 0,C 180,E1 -15208.733,E2 -15208.733} C_VEL
LIN {X 0,Y 317.738,Z 401.785,A -85,B 0,C 180,E1 -15210,E2 -15210} C_VEL
LIN {X 0,Y 317.722,Z 401.564,A -85,B 0,C 180,E1 -15211.268,E2 -15211.268} C_VEL
LIN {X 0,Y 317.751,Z 400.955,A -85,B 0,C 180,E1 -15212.535,E2 -15212.535} C_VEL
LIN {X 0,Y 317.779,Z 399.956,A -85,B 0,C 180,E1 -15213.804,E2 -15213.804} C_VEL
LIN {X 0,Y 317.824,Z 397.698,A -85,B 0,C 180,E1 -15215.685,E2 -15215.685} C_VEL
LIN {X 0,Y 318.077,Z 394.385,A -85,B 0,C 180,E1 -15217.618,E2 -15217.618} C_VEL
LIN {X 0,Y 318.549,Z 390.041,A -85,B 0,C 180,E1 -15219.524,E2 -15219.524} C_VEL
LIN {X 0,Y 319.234,Z 384.509,A -85,B 0,C 180,E1 -15221.428,E2 -15221.428} C_VEL
LIN {X 0,Y 320.265,Z 377.608,A -85,B 0,C 180,E1 -15223.322,E2 -15223.322} C_VEL
LIN {X 0,Y 321.322,Z 370.562,A -85,B 0,C 180,E1 -15224.892,E2 -15224.892} C_VEL
LIN {X 0,Y 322.447,Z 362.066,A -85,B 0,C 180,E1 -15226.46,E2 -15226.46} C_VEL
LIN {X 0,Y 323.902,Z 351.572,A -85,B 0,C 180,E1 -15228.011,E2 -15228.011} C_VEL
LIN {X 0,Y 325.495,Z 339.762,A -85,B 0,C 180,E1 -15229.389,E2 -15229.389} C_VEL
LIN {X 0,Y 326.815,Z 327.869,A -85,B 0,C 180,E1 -15230.454,E2 -15230.454} C_VEL
LIN {X 0,Y 328.021,Z 315.492,A -85,B 0,C 180,E1 -15231.278,E2 -15231.278} C_VEL
LIN {X 0,Y 328.963,Z 302.753,A -85,B 0,C 180,E1 -15231.872,E2 -15231.872} C_VEL
LIN {X 0,Y 329.499,Z 289.31,A -85,B 0,C 180,E1 -15232.247,E2 -15232.247} C_VEL
LIN {X 0,Y 330.591,Z 227.065,A -85,B 0,C 180,E1 -15233.606,E2 -15233.606} C_VEL
LIN {X 0,Y 326.069,Z 199.989,A -85,B 0,C 180,E1 -15234.591,E2 -15234.591} C_VEL
LIN {X 0,Y 324.014,Z 189.274,A -85,B 0,C 180,E1 -15235.027,E2 -15235.027} C_VEL
LIN {X 0,Y 323.477,Z 184.561,A -85,B 0,C 180,E1 -15236.372,E2 -15236.372} C_VEL
LIN {X 0,Y 321.339,Z 174.028,A -85,B 0,C 180,E1 -15239.537,E2 -15239.537} C_VEL
LIN {X 0,Y 319.56,Z 166.174,A -85,B 0,C 180,E1 -15242.044,E2 -15242.044} C_VEL
LIN {X 0,Y 319.578,Z 166.176,A -85,B 0,C 180,E1 -15245.542,E2 -15245.542} C_VEL
LIN {X 0,Y 319.528,Z 166.182,A -85,B 0,C 180,E1 -15249.662,E2 -15249.662} C_VEL
LIN {X 0,Y 319.52,Z 166.183,A -85,B 0,C 180,E1 -15253.46,E2 -15253.46} C_VEL
LIN {X 0,Y 319.553,Z 166.179,A -85,B 0,C 180,E1 -15257.016,E2 -15257.016} C_VEL
LIN {X 0,Y 319.546,Z 166.183,A -85,B 0,C 180,E1 -15260.371,E2 -15260.371} C_VEL
LIN {X 0,Y 319.58,Z 166.178,A -85,B 0,C 180,E1 -15264.457,E2 -15264.457} C_VEL
LIN {X 0,Y 319.524,Z 166.186,A -85,B 0,C 180,E1 -15268.137,E2 -15268.137} C_VEL
LIN {X 0,Y 319.588,Z 166.175,A -85,B 0,C 180,E1 -15271.598,E2 -15271.598} C_VEL
LIN {X 0,Y 319.582,Z 166.175,A -85,B 0,C 180,E1 -15275.302,E2 -15275.302} C_VEL
LIN {X 0,Y 319.602,Z 166.173,A -85,B 0,C 180,E1 -15279.4,E2 -15279.4} C_VEL
LIN {X 0,Y 319.658,Z 166.165,A -85,B 0,C 180,E1 -15282.073,E2 -15282.073} C_VEL
LIN {X 0,Y 319.732,Z 166.156,A -85,B 0,C 180,E1 -15286.008,E2 -15286.008} C_VEL
LIN {X 0,Y 319.752,Z 166.155,A -85,B 0,C 180,E1 -15289.873,E2 -15289.873} C_VEL
LIN {X 0,Y 319.912,Z 166.131,A -85,B 0,C 180,E1 -15292.426,E2 -15292.426} C_VEL
LIN {X 0,Y 319.744,Z 166.154,A -85,B 0,C 180,E1 -15294.956,E2 -15294.956} C_VEL
LIN {X 0,Y 319.99,Z 166.126,A -85,B 0,C 180,E1 -15297.482,E2 -15297.482} C_VEL
LIN {X 0,Y 320.132,Z 166.103,A -85,B 0,C 180,E1 -15300,E2 -15300} C_VEL
LIN {X 0,Y 319.991,Z 166.124,A -85,B 0,C 180,E1 -15302.518,E2 -15302.518} C_VEL
LIN {X 0,Y 319.924,Z 166.128,A -85,B 0,C 180,E1 -15306.51,E2 -15306.51} C_VEL
LIN {X 0,Y 319.838,Z 166.146,A -85,B 0,C 180,E1 -15308.848,E2 -15308.848} C_VEL
LIN {X 0,Y 319.682,Z 166.163,A -85,B 0,C 180,E1 -15312.7,E2 -15312.7} C_VEL
LIN {X 0,Y 319.7,Z 166.16,A -85,B 0,C 180,E1 -15315.296,E2 -15315.296} C_VEL
LIN {X 0,Y 319.675,Z 166.163,A -85,B 0,C 180,E1 -15319.255,E2 -15319.255} C_VEL
LIN {X 0,Y 319.57,Z 166.174,A -85,B 0,C 180,E1 -15323.32,E2 -15323.32} C_VEL
LIN {X 0,Y 319.635,Z 166.169,A -85,B 0,C 180,E1 -15326.088,E2 -15326.088} C_VEL
LIN {X 0,Y 319.59,Z 166.174,A -85,B 0,C 180,E1 -15328.934,E2 -15328.934} C_VEL
LIN {X 0,Y 319.532,Z 166.181,A -85,B 0,C 180,E1 -15331.862,E2 -15331.862} C_VEL
LIN {X 0,Y 319.58,Z 166.174,A -85,B 0,C 180,E1 -15335.543,E2 -15335.543} C_VEL
LIN {X 0,Y 319.573,Z 166.18,A -85,B 0,C 180,E1 -15338.008,E2 -15338.008} C_VEL
LIN {X 0,Y 319.526,Z 166.183,A -85,B 0,C 180,E1 -15341.597,E2 -15341.597} C_VEL
LIN {X 0,Y 319.489,Z 166.185,A -85,B 0,C 180,E1 -15345.258,E2 -15345.258} C_VEL
LIN {X 0,Y 319.529,Z 166.181,A -85,B 0,C 180,E1 -15348.712,E2 -15348.712} C_VEL
LIN {X 0,Y 319.562,Z 166.178,A -85,B 0,C 180,E1 -15352.348,E2 -15352.348} C_VEL
LIN {X 0,Y 319.561,Z 166.18,A -85,B 0,C 180,E1 -15355.124,E2 -15355.124} C_VEL
LIN {X 0,Y 319.572,Z 166.18,A -85,B 0,C 180,E1 -15359.058,E2 -15359.058} C_VEL
LIN {X 0,Y 319.62,Z 166.223,A -85,B 0,C 180,E1 -15361.625,E2 -15361.625} C_VEL
LIN {X 0,Y 321.858,Z 176.327,A -85,B 0,C 180,E1 -15364.864,E2 -15364.864} C_VEL
LIN {X 0,Y 328.287,Z 193.215,A -85,B 0,C 180,E1 -15365.792,E2 -15365.792} C_VEL
LIN {X 0,Y 331.118,Z 208.127,A -85,B 0,C 180,E1 -15366.361,E2 -15366.361} C_VEL
LIN {X 0,Y 329.472,Z 283.047,A -85,B 0,C 180,E1 -15367.999,E2 -15367.999} C_VEL
LIN {X 0,Y 328.751,Z 296.462,A -85,B 0,C 180,E1 -15368.525,E2 -15368.525} C_VEL
LIN {X 0,Y 327.813,Z 309.237,A -85,B 0,C 180,E1 -15369.284,E2 -15369.284} C_VEL
LIN {X 0,Y 326.714,Z 320.577,A -85,B 0,C 180,E1 -15370.196,E2 -15370.196} C_VEL
LIN {X 0,Y 325.312,Z 332.232,A -85,B 0,C 180,E1 -15371.418,E2 -15371.418} C_VEL
LIN {X 0,Y 324.05,Z 342.664,A -85,B 0,C 180,E1 -15372.809,E2 -15372.809} C_VEL
LIN {X 0,Y 322.899,Z 351.235,A -85,B 0,C 180,E1 -15374.213,E2 -15374.213} C_VEL
LIN {X 0,Y 321.599,Z 359.111,A -85,B 0,C 180,E1 -15375.768,E2 -15375.768} C_VEL
LIN {X 0,Y 320.44,Z 366.805,A -85,B 0,C 180,E1 -15377.652,E2 -15377.652} C_VEL
LIN {X 0,Y 319.372,Z 373.867,A -85,B 0,C 180,E1 -15379.86,E2 -15379.86} C_VEL
LIN {X 0,Y 318.678,Z 378.571,A -85,B 0,C 180,E1 -15381.758,E2 -15381.758} C_VEL
LIN {X 0,Y 318.316,Z 382.168,A -85,B 0,C 180,E1 -15383.662,E2 -15383.662} C_VEL
LIN {X 0,Y 318.124,Z 384.027,A -85,B 0,C 180,E1 -15384.93,E2 -15384.93} C_VEL
LIN {X 0,Y 317.976,Z 385.426,A -85,B 0,C 180,E1 -15386.198,E2 -15386.198} C_VEL
LIN {X 0,Y 317.768,Z 387.035,A -85,B 0,C 180,E1 -15388.733,E2 -15388.733} C_VEL
LIN {X 0,Y 317.744,Z 387.267,A -85,B 0,C 180,E1 -15390,E2 -15390} C_VEL
LIN {X 0,Y 317.767,Z 387.076,A -85,B 0,C 180,E1 -15391.267,E2 -15391.267} C_VEL
LIN {X 0,Y 317.972,Z 385.52,A -85,B 0,C 180,E1 -15393.802,E2 -15393.802} C_VEL
LIN {X 0,Y 318.111,Z 384.162,A -85,B 0,C 180,E1 -15395.07,E2 -15395.07} C_VEL
LIN {X 0,Y 318.413,Z 381.294,A -85,B 0,C 180,E1 -15396.972,E2 -15396.972} C_VEL
LIN {X 0,Y 318.869,Z 377.402,A -85,B 0,C 180,E1 -15398.875,E2 -15398.875} C_VEL
LIN {X 0,Y 319.616,Z 372.38,A -85,B 0,C 180,E1 -15400.772,E2 -15400.772} C_VEL
LIN {X 0,Y 320.593,Z 366.057,A -85,B 0,C 180,E1 -15402.663,E2 -15402.663} C_VEL
LIN {X 0,Y 321.797,Z 358.143,A -85,B 0,C 180,E1 -15404.546,E2 -15404.546} C_VEL
LIN {X 0,Y 323.336,Z 348.296,A -85,B 0,C 180,E1 -15406.413,E2 -15406.413} C_VEL
LIN {X 0,Y 324.665,Z 337.963,A -85,B 0,C 180,E1 -15407.967,E2 -15407.967} C_VEL
LIN {X 0,Y 325.917,Z 327.726,A -85,B 0,C 180,E1 -15409.199,E2 -15409.199} C_VEL
LIN {X 0,Y 327.194,Z 316.522,A -85,B 0,C 180,E1 -15410.265,E2 -15410.265} C_VEL
LIN {X 0,Y 328.343,Z 303.893,A -85,B 0,C 180,E1 -15411.174,E2 -15411.174} C_VEL
LIN {X 0,Y 329.084,Z 291.231,A -85,B 0,C 180,E1 -15411.822,E2 -15411.822} C_VEL
LIN {X 0,Y 329.71,Z 278.199,A -85,B 0,C 180,E1 -15412.232,E2 -15412.232} C_VEL
LIN {X 0,Y 331.121,Z 207.759,A -85,B 0,C 180,E1 -15413.761,E2 -15413.761} C_VEL
LIN {X 0,Y 327.948,Z 191.871,A -85,B 0,C 180,E1 -15414.38,E2 -15414.38} C_VEL
LIN {X 0,Y 321.8,Z 176.083,A -85,B 0,C 180,E1 -15415.301,E2 -15415.301} C_VEL
LIN {X 0,Y 319.948,Z 167.616,A -85,B 0,C 180,E1 -15418.033,E2 -15418.033} C_VEL
LIN {X 0,Y 319.606,Z 166.175,A -85,B 0,C 180,E1 -15418.53,E2 -15418.53} C_VEL
LIN {X 0,Y 319.533,Z 166.183,A -85,B 0,C 180,E1 -15421.861,E2 -15421.861} C_VEL
LIN {X 0,Y 319.569,Z 166.176,A -85,B 0,C 180,E1 -15423.452,E2 -15423.452} C_VEL
LIN {X 0,Y 318.863,Z 166.265,A -85,B 0,C 180,E1 -15424.503,E2 -15424.503} C_VEL
LIN {X 0,Y 316.029,Z 166.62,A -85,B 0,C 180,E1 -15426.215,E2 -15426.215} C_VEL
LIN {X 0,Y 313.641,Z 166.918,A -85,B 0,C 180,E1 -15427.602,E2 -15427.602} C_VEL
LIN {X 0,Y 312.599,Z 167.046,A -85,B 0,C 180,E1 -15428.676,E2 -15428.676} C_VEL
LIN {X 0,Y 312.503,Z 167.056,A -85,B 0,C 180,E1 -15429.039,E2 -15429.039} C_VEL
LIN {X 0,Y 312.491,Z 167.061,A -85,B 0,C 180,E1 -15432.431,E2 -15432.431} C_VEL
LIN {X 0,Y 312.458,Z 167.065,A -85,B 0,C 180,E1 -15436.035,E2 -15436.035} C_VEL
LIN {X 0,Y 312.504,Z 167.059,A -85,B 0,C 180,E1 -15439.874,E2 -15439.874} C_VEL
LIN {X 0,Y 312.537,Z 167.05,A -85,B 0,C 180,E1 -15442.616,E2 -15442.616} C_VEL
LIN {X 0,Y 312.519,Z 167.051,A -85,B 0,C 180,E1 -15446.311,E2 -15446.311} C_VEL
LIN {X 0,Y 312.545,Z 167.05,A -85,B 0,C 180,E1 -15450.35,E2 -15450.35} C_VEL
LIN {X 0,Y 312.603,Z 167.045,A -85,B 0,C 180,E1 -15454.064,E2 -15454.064} C_VEL
LIN {X 0,Y 312.587,Z 167.045,A -85,B 0,C 180,E1 -15457.529,E2 -15457.529} C_VEL
LIN {X 0,Y 312.638,Z 167.041,A -85,B 0,C 180,E1 -15461.656,E2 -15461.656} C_VEL
LIN {X 0,Y 312.693,Z 167.033,A -85,B 0,C 180,E1 -15465.686,E2 -15465.686} C_VEL
LIN {X 0,Y 312.701,Z 167.03,A -85,B 0,C 180,E1 -15469.642,E2 -15469.642} C_VEL
LIN {X 0,Y 312.865,Z 167.006,A -85,B 0,C 180,E1 -15472.254,E2 -15472.254} C_VEL
LIN {X 0,Y 312.715,Z 167.033,A -85,B 0,C 180,E1 -15474.842,E2 -15474.842} C_VEL
LIN {X 0,Y 312.988,Z 166.994,A -85,B 0,C 180,E1 -15478.713,E2 -15478.713} C_VEL
LIN {X 0,Y 312.99,Z 166.996,A -85,B 0,C 180,E1 -15481.287,E2 -15481.287} C_VEL
LIN {X 0,Y 312.714,Z 167.026,A -85,B 0,C 180,E1 -15485.158,E2 -15485.158} C_VEL
LIN {X 0,Y 312.865,Z 167.008,A -85,B 0,C 180,E1 -15487.746,E2 -15487.746} C_VEL
LIN {X 0,Y 312.668,Z 167.034,A -85,B 0,C 180,E1 -15491.671,E2 -15491.671} C_VEL
LIN {X 0,Y 312.699,Z 167.032,A -85,B 0,C 180,E1 -15494.888,E2 -15494.888} C_VEL
LIN {X 0,Y 312.608,Z 167.038,A -85,B 0,C 180,E1 -15499.225,E2 -15499.225} C_VEL
LIN {X 0,Y 312.525,Z 167.053,A -85,B 0,C 180,E1 -15502.781,E2 -15502.781} C_VEL
LIN {X 0,Y 312.601,Z 167.044,A -85,B 0,C 180,E1 -15505.935,E2 -15505.935} C_VEL
LIN {X 0,Y 312.537,Z 167.054,A -85,B 0,C 180,E1 -15509.651,E2 -15509.651} C_VEL
LIN {X 0,Y 312.519,Z 167.057,A -85,B 0,C 180,E1 -15513.689,E2 -15513.689} C_VEL
LIN {X 0,Y 312.519,Z 167.057,A -85,B 0,C 180,E1 -15517.386,E2 -15517.386} C_VEL
LIN {X 0,Y 312.489,Z 167.058,A -85,B 0,C 180,E1 -15520.709,E2 -15520.709} C_VEL
LIN {X 0,Y 312.451,Z 167.062,A -85,B 0,C 180,E1 -15524.21,E2 -15524.21} C_VEL
LIN {X 0,Y 312.455,Z 167.063,A -85,B 0,C 180,E1 -15527.925,E2 -15527.925} C_VEL
LIN {X 0,Y 312.484,Z 167.059,A -85,B 0,C 180,E1 -15531.923,E2 -15531.923} C_VEL
LIN {X 0,Y 312.531,Z 167.053,A -85,B 0,C 180,E1 -15534.22,E2 -15534.22} C_VEL
LIN {X 0,Y 312.545,Z 167.129,A -85,B 0,C 180,E1 -15537.504,E2 -15537.504} C_VEL
LIN {X 0,Y 314.83,Z 177.425,A -85,B 0,C 180,E1 -15540.81,E2 -15540.81} C_VEL
LIN {X 0,Y 316.94,Z 188.118,A -85,B 0,C 180,E1 -15544.072,E2 -15544.072} C_VEL
LIN {X 0,Y 317.071,Z 189.089,A -85,B 0,C 180,E1 -15544.357,E2 -15544.357} C_VEL
LIN {X 0,Y 318.879,Z 197.369,A -85,B 0,C 180,E1 -15544.732,E2 -15544.732} C_VEL
LIN {X 0,Y 323.109,Z 221.422,A -85,B 0,C 180,E1 -15545.659,E2 -15545.659} C_VEL
LIN {X 0,Y 324.223,Z 228.754,A -85,B 0,C 180,E1 -15545.921,E2 -15545.921} C_VEL
LIN {X 0,Y 322.657,Z 297.603,A -85,B 0,C 180,E1 -15547.467,E2 -15547.467} C_VEL
LIN {X 0,Y 321.753,Z 310.771,A -85,B 0,C 180,E1 -15547.992,E2 -15547.992} C_VEL
LIN {X 0,Y 320.746,Z 322.879,A -85,B 0,C 180,E1 -15548.721,E2 -15548.721} C_VEL
LIN {X 0,Y 319.401,Z 335.1,A -85,B 0,C 180,E1 -15549.723,E2 -15549.723} C_VEL
LIN {X 0,Y 317.857,Z 346.671,A -85,B 0,C 180,E1 -15550.966,E2 -15550.966} C_VEL
LIN {X 0,Y 316.399,Z 357.092,A -85,B 0,C 180,E1 -15552.384,E2 -15552.384} C_VEL
LIN {X 0,Y 315.099,Z 366.273,A -85,B 0,C 180,E1 -15553.938,E2 -15553.938} C_VEL
LIN {X 0,Y 313.781,Z 374.852,A -85,B 0,C 180,E1 -15555.737,E2 -15555.737} C_VEL
LIN {X 0,Y 312.557,Z 382.275,A -85,B 0,C 180,E1 -15557.666,E2 -15557.666} C_VEL
LIN {X 0,Y 311.727,Z 388.24,A -85,B 0,C 180,E1 -15559.609,E2 -15559.609} C_VEL
LIN {X 0,Y 311.156,Z 392.954,A -85,B 0,C 180,E1 -15561.558,E2 -15561.558} C_VEL
LIN {X 0,Y 310.822,Z 396.556,A -85,B 0,C 180,E1 -15563.509,E2 -15563.509} C_VEL
LIN {X 0,Y 310.696,Z 398.414,A -85,B 0,C 180,E1 -15564.809,E2 -15564.809} C_VEL
LIN {X 0,Y 310.691,Z 399.809,A -85,B 0,C 180,E1 -15566.109,E2 -15566.109} C_VEL
LIN {X 0,Y 310.673,Z 400.804,A -85,B 0,C 180,E1 -15567.407,E2 -15567.407} C_VEL
LIN {X 0,Y 310.638,Z 401.41,A -85,B 0,C 180,E1 -15568.704,E2 -15568.704} C_VEL
LIN {X 0,Y 310.65,Z 401.623,A -85,B 0,C 180,E1 -15570,E2 -15570} C_VEL
LIN {X 0,Y 310.638,Z 401.402,A -85,B 0,C 180,E1 -15571.296,E2 -15571.296} C_VEL
LIN {X 0,Y 310.673,Z 400.792,A -85,B 0,C 180,E1 -15572.593,E2 -15572.593} C_VEL
LIN {X 0,Y 310.692,Z 399.793,A -85,B 0,C 180,E1 -15573.891,E2 -15573.891} C_VEL
LIN {X 0,Y 310.723,Z 397.813,A -85,B 0,C 180,E1 -15575.614,E2 -15575.614} C_VEL
LIN {X 0,Y 311.02,Z 394.221,A -85,B 0,C 180,E1 -15577.792,E2 -15577.792} C_VEL
LIN {X 0,Y 311.508,Z 389.877,A -85,B 0,C 180,E1 -15579.742,E2 -15579.742} C_VEL
LIN {X 0,Y 312.225,Z 384.344,A -85,B 0,C 180,E1 -15581.688,E2 -15581.688} C_VEL
LIN {X 0,Y 313.327,Z 377.444,A -85,B 0,C 180,E1 -15583.622,E2 -15583.622} C_VEL
LIN {X 0,Y 314.41,Z 370.396,A -85,B 0,C 180,E1 -15585.227,E2 -15585.227} C_VEL
LIN {X 0,Y 315.624,Z 361.901,A -85,B 0,C 180,E1 -15586.826,E2 -15586.826} C_VEL
LIN {X 0,Y 317.132,Z 351.406,A -85,B 0,C 180,E1 -15588.409,E2 -15588.409} C_VEL
LIN {X 0,Y 318.816,Z 339.596,A -85,B 0,C 180,E1 -15589.811,E2 -15589.811} C_VEL
LIN {X 0,Y 320.174,Z 327.701,A -85,B 0,C 180,E1 -15590.897,E2 -15590.897} C_VEL
LIN {X 0,Y 321.402,Z 315.321,A -85,B 0,C 180,E1 -15591.738,E2 -15591.738} C_VEL
LIN {X 0,Y 322.394,Z 302.58,A -85,B 0,C 180,E1 -15592.342,E2 -15592.342} C_VEL
LIN {X 0,Y 322.935,Z 289.127,A -85,B 0,C 180,E1 -15592.724,E2 -15592.724} C_VEL
LIN {X 0,Y 324.073,Z 227.924,A -85,B 0,C 180,E1 -15594.086,E2 -15594.086} C_VEL
LIN {X 0,Y 319.462,Z 200.379,A -85,B 0,C 180,E1 -15595.12,E2 -15595.12} C_VEL
LIN {X 0,Y 317.096,Z 189.282,A -85,B 0,C 180,E1 -15595.591,E2 -15595.591} C_VEL
LIN {X 0,Y 315.431,Z 180.333,A -85,B 0,C 180,E1 -15598.259,E2 -15598.259} C_VEL
LIN {X 0,Y 313.212,Z 170.091,A -85,B 0,C 180,E1 -15601.497,E2 -15601.497} C_VEL
LIN {X 0,Y 312.544,Z 167.051,A -85,B 0,C 180,E1 -15602.495,E2 -15602.495} C_VEL
LIN {X 0,Y 312.534,Z 167.054,A -85,B 0,C 180,E1 -15605.949,E2 -15605.949} C_VEL
LIN {X 0,Y 312.455,Z 167.064,A -85,B 0,C 180,E1 -15610.114,E2 -15610.114} C_VEL
LIN {X 0,Y 312.457,Z 167.063,A -85,B 0,C 180,E1 -15613.965,E2 -15613.965} C_VEL
LIN {X 0,Y 312.483,Z 167.059,A -85,B 0,C 180,E1 -15617.919,E2 -15617.919} C_VEL
LIN {X 0,Y 312.498,Z 167.058,A -85,B 0,C 180,E1 -15620.971,E2 -15620.971} C_VEL
LIN {X 0,Y 312.532,Z 167.056,A -85,B 0,C 180,E1 -15624.22,E2 -15624.22} C_VEL
LIN {X 0,Y 312.501,Z 167.056,A -85,B 0,C 180,E1 -15627.333,E2 -15627.333} C_VEL
LIN {X 0,Y 312.519,Z 167.054,A -85,B 0,C 180,E1 -15631.287,E2 -15631.287} C_VEL
LIN {X 0,Y 312.553,Z 167.05,A -85,B 0,C 180,E1 -15634.708,E2 -15634.708} C_VEL
LIN {X 0,Y 312.563,Z 167.048,A -85,B 0,C 180,E1 -15637.527,E2 -15637.527} C_VEL
LIN {X 0,Y 312.638,Z 167.041,A -85,B 0,C 180,E1 -15641.656,E2 -15641.656} C_VEL
LIN {X 0,Y 312.694,Z 167.036,A -85,B 0,C 180,E1 -15645.686,E2 -15645.686} C_VEL
LIN {X 0,Y 312.698,Z 167.036,A -85,B 0,C 180,E1 -15649.642,E2 -15649.642} C_VEL
LIN {X 0,Y 312.853,Z 167.011,A -85,B 0,C 180,E1 -15652.254,E2 -15652.254} C_VEL
LIN {X 0,Y 312.714,Z 167.029,A -85,B 0,C 180,E1 -15654.842,E2 -15654.842} C_VEL
LIN {X 0,Y 312.99,Z 166.995,A -85,B 0,C 180,E1 -15658.713,E2 -15658.713} C_VEL
LIN {X 0,Y 312.989,Z 166.999,A -85,B 0,C 180,E1 -15661.287,E2 -15661.287} C_VEL
LIN {X 0,Y 312.712,Z 167.03,A -85,B 0,C 180,E1 -15665.158,E2 -15665.158} C_VEL
LIN {X 0,Y 312.856,Z 167.012,A -85,B 0,C 180,E1 -15667.746,E2 -15667.746} C_VEL
LIN {X 0,Y 312.669,Z 167.032,A -85,B 0,C 180,E1 -15671.671,E2 -15671.671} C_VEL
LIN {X 0,Y 312.7,Z 167.035,A -85,B 0,C 180,E1 -15674.888,E2 -15674.888} C_VEL
LIN {X 0,Y 312.631,Z 167.041,A -85,B 0,C 180,E1 -15679.237,E2 -15679.237} C_VEL
LIN {X 0,Y 312.546,Z 167.052,A -85,B 0,C 180,E1 -15682.789,E2 -15682.789} C_VEL
LIN {X 0,Y 312.603,Z 167.045,A -85,B 0,C 180,E1 -15685.936,E2 -15685.936} C_VEL
LIN {X 0,Y 312.546,Z 167.051,A -85,B 0,C 180,E1 -15689.65,E2 -15689.65} C_VEL
LIN {X 0,Y 312.52,Z 167.055,A -85,B 0,C 180,E1 -15693.689,E2 -15693.689} C_VEL
LIN {X 0,Y 312.537,Z 167.052,A -85,B 0,C 180,E1 -15697.384,E2 -15697.384} C_VEL
LIN {X 0,Y 312.49,Z 167.058,A -85,B 0,C 180,E1 -15700.709,E2 -15700.709} C_VEL
LIN {X 0,Y 312.452,Z 167.064,A -85,B 0,C 180,E1 -15704.21,E2 -15704.21} C_VEL
LIN {X 0,Y 312.485,Z 167.061,A -85,B 0,C 180,E1 -15707.919,E2 -15707.919} C_VEL
LIN {X 0,Y 312.536,Z 167.055,A -85,B 0,C 180,E1 -15711.911,E2 -15711.911} C_VEL
LIN {X 0,Y 312.508,Z 167.058,A -85,B 0,C 180,E1 -15715.79,E2 -15715.79} C_VEL
LIN {X 0,Y 312.525,Z 167.058,A -85,B 0,C 180,E1 -15718.854,E2 -15718.854} C_VEL
LIN {X 0,Y 312.571,Z 167.068,A -85,B 0,C 180,E1 -15721.138,E2 -15721.138} C_VEL
LIN {X 0,Y 314.706,Z 176.535,A -85,B 0,C 180,E1 -15724.252,E2 -15724.252} C_VEL
LIN {X 0,Y 322.014,Z 195.248,A -85,B 0,C 180,E1 -15725.334,E2 -15725.334} C_VEL
LIN {X 0,Y 324.621,Z 208.692,A -85,B 0,C 180,E1 -15725.867,E2 -15725.867} C_VEL
LIN {X 0,Y 323.013,Z 281.783,A -85,B 0,C 180,E1 -15727.493,E2 -15727.493} C_VEL
LIN {X 0,Y 322.323,Z 294.338,A -85,B 0,C 180,E1 -15727.948,E2 -15727.948} C_VEL
LIN {X 0,Y 321.411,Z 307.15,A -85,B 0,C 180,E1 -15728.683,E2 -15728.683} C_VEL
LIN {X 0,Y 320.215,Z 319.006,A -85,B 0,C 180,E1 -15729.609,E2 -15729.609} C_VEL
LIN {X 0,Y 318.939,Z 329.763,A -85,B 0,C 180,E1 -15730.699,E2 -15730.699} C_VEL
LIN {X 0,Y 317.643,Z 339.651,A -85,B 0,C 180,E1 -15731.955,E2 -15731.955} C_VEL
LIN {X 0,Y 316.384,Z 349.624,A -85,B 0,C 180,E1 -15733.547,E2 -15733.547} C_VEL
LIN {X 0,Y 314.712,Z 359.276,A -85,B 0,C 180,E1 -15735.45,E2 -15735.45} C_VEL
LIN {X 0,Y 313.513,Z 366.969,A -85,B 0,C 180,E1 -15737.375,E2 -15737.375} C_VEL
LIN {X 0,Y 312.367,Z 374.031,A -85,B 0,C 180,E1 -15739.631,E2 -15739.631} C_VEL
LIN {X 0,Y 311.657,Z 378.734,A -85,B 0,C 180,E1 -15741.571,E2 -15741.571} C_VEL
LIN {X 0,Y 311.263,Z 382.331,A -85,B 0,C 180,E1 -15743.518,E2 -15743.518} C_VEL
LIN {X 0,Y 311.058,Z 384.19,A -85,B 0,C 180,E1 -15744.815,E2 -15744.815} C_VEL
LIN {X 0,Y 310.913,Z 385.588,A -85,B 0,C 180,E1 -15746.112,E2 -15746.112} C_VEL
LIN {X 0,Y 310.682,Z 387.197,A -85,B 0,C 180,E1 -15748.704,E2 -15748.704} C_VEL
LIN {X 0,Y 310.656,Z 387.429,A -85,B 0,C 180,E1 -15750,E2 -15750} C_VEL
LIN {X 0,Y 310.682,Z 387.237,A -85,B 0,C 180,E1 -15751.296,E2 -15751.296} C_VEL
LIN {X 0,Y 310.908,Z 385.681,A -85,B 0,C 180,E1 -15753.888,E2 -15753.888} C_VEL
LIN {X 0,Y 311.042,Z 384.324,A -85,B 0,C 180,E1 -15755.185,E2 -15755.185} C_VEL
LIN {X 0,Y 311.358,Z 381.454,A -85,B 0,C 180,E1 -15757.131,E2 -15757.131} C_VEL
LIN {X 0,Y 311.849,Z 377.563,A -85,B 0,C 180,E1 -15759.077,E2 -15759.077} C_VEL
LIN {X 0,Y 312.619,Z 372.541,A -85,B 0,C 180,E1 -15761.016,E2 -15761.016} C_VEL
LIN {X 0,Y 313.637,Z 366.218,A -85,B 0,C 180,E1 -15762.949,E2 -15762.949} C_VEL
LIN {X 0,Y 314.942,Z 358.302,A -85,B 0,C 180,E1 -15764.87,E2 -15764.87} C_VEL
LIN {X 0,Y 316.529,Z 348.455,A -85,B 0,C 180,E1 -15766.777,E2 -15766.777} C_VEL
LIN {X 0,Y 317.746,Z 339.291,A -85,B 0,C 180,E1 -15768.205,E2 -15768.205} C_VEL
LIN {X 0,Y 319.214,Z 327.883,A -85,B 0,C 180,E1 -15769.618,E2 -15769.618} C_VEL
LIN {X 0,Y 320.538,Z 316.678,A -85,B 0,C 180,E1 -15770.704,E2 -15770.704} C_VEL
LIN {X 0,Y 321.748,Z 304.046,A -85,B 0,C 180,E1 -15771.629,E2 -15771.629} C_VEL
LIN {X 0,Y 322.529,Z 291.38,A -85,B 0,C 180,E1 -15772.289,E2 -15772.289} C_VEL
LIN {X 0,Y 323.173,Z 278.34,A -85,B 0,C 180,E1 -15772.706,E2 -15772.706} C_VEL
LIN {X 0,Y 324.622,Z 208.375,A -85,B 0,C 180,E1 -15774.255,E2 -15774.255} C_VEL
LIN {X 0,Y 321.724,Z 194.217,A -85,B 0,C 180,E1 -15774.83,E2 -15774.83} C_VEL
LIN {X 0,Y 314.65,Z 176.263,A -85,B 0,C 180,E1 -15775.915,E2 -15775.915} C_VEL
LIN {X 0,Y 312.544,Z 167.056,A -85,B 0,C 180,E1 -15778.994,E2 -15778.994} C_VEL
LIN {X 0,Y 312.505,Z 167.061,A -85,B 0,C 180,E1 -15782.666,E2 -15782.666} C_VEL
LIN {X 0,Y 312.536,Z 167.053,A -85,B 0,C 180,E1 -15785.949,E2 -15785.949} C_VEL
LIN {X 0,Y 312.503,Z 167.056,A -85,B 0,C 180,E1 -15789.039,E2 -15789.039} C_VEL
LIN {X 0,Y 311.804,Z 167.146,A -85,B 0,C 180,E1 -15790.116,E2 -15790.116} C_VEL
LIN {X 0,Y 308.937,Z 167.502,A -85,B 0,C 180,E1 -15791.867,E2 -15791.867} C_VEL
LIN {X 0,Y 306.521,Z 167.804,A -85,B 0,C 180,E1 -15793.287,E2 -15793.287} C_VEL
LIN {X 0,Y 305.479,Z 167.933,A -85,B 0,C 180,E1 -15794.387,E2 -15794.387} C_VEL
LIN {X 0,Y 305.391,Z 167.941,A -85,B 0,C 180,E1 -15794.76,E2 -15794.76} C_VEL
LIN {X 0,Y 305.441,Z 167.937,A -85,B 0,C 180,E1 -15798.143,E2 -15798.143} C_VEL
LIN {X 0,Y 305.495,Z 167.93,A -85,B 0,C 180,E1 -15801.6,E2 -15801.6} C_VEL
LIN {X 0,Y 305.462,Z 167.932,A -85,B 0,C 180,E1 -15804.887,E2 -15804.887} C_VEL
LIN {X 0,Y 305.452,Z 167.935,A -85,B 0,C 180,E1 -15808.355,E2 -15808.355} C_VEL
LIN {X 0,Y 305.52,Z 167.925,A -85,B 0,C 180,E1 -15811.114,E2 -15811.114} C_VEL
LIN {X 0,Y 305.571,Z 167.921,A -85,B 0,C 180,E1 -15814.088,E2 -15814.088} C_VEL
LIN {X 0,Y 305.5,Z 167.924,A -85,B 0,C 180,E1 -15818.403,E2 -15818.403} C_VEL
LIN {X 0,Y 305.59,Z 167.921,A -85,B 0,C 180,E1 -15821.218,E2 -15821.218} C_VEL
LIN {X 0,Y 305.648,Z 167.909,A -85,B 0,C 180,E1 -15825.349,E2 -15825.349} C_VEL
